LIN {X 0,Y 425.746,Z 248.042,A -85,B 0,C 180,E1 19809.734,E2 19809.734} C_VEL
LIN {X 0,Y 425.285,Z 246.258,A -85,B 0,C 180,E1 19809.199,E2 19809.199} C_VEL
LIN {X 0,Y 425.24,Z 246.07,A -85,B 0,C 180,E1 19805.532,E2 19805.532} C_VEL
LIN {X 0,Y 425.24,Z 246.073,A -85,B 0,C 180,E1 19801.616,E2 19801.616} C_VEL
LIN {X 0,Y 425.257,Z 246.076,A -85,B 0,C 180,E1 19797.978,E2 19797.978} C_VEL
LIN {X 0,Y 425.284,Z 246.063,A -85,B 0,C 180,E1 19794.197,E2 19794.197} C_VEL
LIN {X 0,Y 425.27,Z 246.064,A -85,B 0,C 180,E1 19790.527,E2 19790.527} C_VEL
LIN {X 0,Y 425.247,Z 246.076,A -85,B 0,C 180,E1 19786.749,E2 19786.749} C_VEL
LIN {X 0,Y 425.238,Z 246.075,A -85,B 0,C 180,E1 19783.048,E2 19783.048} C_VEL
LIN {X 0,Y 425.242,Z 246.067,A -85,B 0,C 180,E1 19779.204,E2 19779.204} C_VEL
LIN {X 0,Y 425.274,Z 246.074,A -85,B 0,C 180,E1 19775.556,E2 19775.556} C_VEL
LIN {X 0,Y 425.312,Z 246.344,A -85,B 0,C 180,E1 19773.47,E2 19773.47} C_VEL
LIN {X 0,Y 426.471,Z 249.444,A -85,B 0,C 180,E1 19772.644,E2 19772.644} C_VEL
LIN {X 0,Y 428.836,Z 251.992,A -85,B 0,C 180,E1 19771.751,E2 19771.751} C_VEL
LIN {X 0,Y 430.464,Z 255.45,A -85,B 0,C 180,E1 19770.958,E2 19770.958} C_VEL
LIN {X 0,Y 432.236,Z 257.496,A -85,B 0,C 180,E1 19770.328,E2 19770.328} C_VEL
LIN {X 0,Y 434.45,Z 261.508,A -85,B 0,C 180,E1 19769.428,E2 19769.428} C_VEL
LIN {X 0,Y 435.82,Z 263.65,A -85,B 0,C 180,E1 19768.922,E2 19768.922} C_VEL
LIN {X 0,Y 439.262,Z 269.551,A -85,B 0,C 180,E1 19767.662,E2 19767.662} C_VEL
LIN {X 0,Y 443.697,Z 276.942,A -85,B 0,C 180,E1 19766.178,E2 19766.178} C_VEL
LIN {X 0,Y 451.348,Z 291.113,A -85,B 0,C 180,E1 19763.738,E2 19763.738} C_VEL
LIN {X 0,Y 458.605,Z 305.629,A -85,B 0,C 180,E1 19761.584,E2 19761.584} C_VEL
LIN {X 0,Y 462.483,Z 314.322,A -85,B 0,C 180,E1 19760.454,E2 19760.454} C_VEL
LIN {X 0,Y 461.558,Z 326.532,A -85,B 0,C 180,E1 19759.768,E2 19759.768} C_VEL
LIN {X 0,Y 463.161,Z 344.572,A -85,B 0,C 180,E1 19759.232,E2 19759.232} C_VEL
LIN {X 0,Y 458.976,Z 547.408,A -85,B 0,C 180,E1 19755.792,E2 19755.792} C_VEL
LIN {X 0,Y 456.721,Z 660.808,A -85,B 0,C 180,E1 19753.907,E2 19753.907} C_VEL
LIN {X 0,Y 455.349,Z 683.856,A -85,B 0,C 180,E1 19753.332,E2 19753.332} C_VEL
LIN {X 0,Y 453.601,Z 706.683,A -85,B 0,C 180,E1 19752.542,E2 19752.542} C_VEL
LIN {X 0,Y 451.584,Z 727.107,A -85,B 0,C 180,E1 19751.621,E2 19751.621} C_VEL
LIN {X 0,Y 449.041,Z 749.414,A -85,B 0,C 180,E1 19750.385,E2 19750.385} C_VEL
LIN {X 0,Y 446.38,Z 769.931,A -85,B 0,C 180,E1 19749.005,E2 19749.005} C_VEL
LIN {X 0,Y 443.463,Z 790.74,A -85,B 0,C 180,E1 19747.335,E2 19747.335} C_VEL
LIN {X 0,Y 440.606,Z 810.204,A -85,B 0,C 180,E1 19745.514,E2 19745.514} C_VEL
LIN {X 0,Y 437.767,Z 828.343,A -85,B 0,C 180,E1 19743.523,E2 19743.523} C_VEL
LIN {X 0,Y 434.981,Z 846.538,A -85,B 0,C 180,E1 19741.23,E2 19741.23} C_VEL
LIN {X 0,Y 432.58,Z 862.117,A -85,B 0,C 180,E1 19738.96,E2 19738.96} C_VEL
LIN {X 0,Y 430.192,Z 878.511,A -85,B 0,C 180,E1 19736.204,E2 19736.204} C_VEL
LIN {X 0,Y 428.326,Z 892.284,A -85,B 0,C 180,E1 19733.525,E2 19733.525} C_VEL
LIN {X 0,Y 426.985,Z 902.738,A -85,B 0,C 180,E1 19731.136,E2 19731.136} C_VEL
LIN {X 0,Y 425.868,Z 911.603,A -85,B 0,C 180,E1 19728.619,E2 19728.619} C_VEL
LIN {X 0,Y 424.933,Z 920.642,A -85,B 0,C 180,E1 19725.558,E2 19725.558} C_VEL
LIN {X 0,Y 424.39,Z 927.376,A -85,B 0,C 180,E1 19722.74,E2 19722.74} C_VEL
LIN {X 0,Y 424.071,Z 933.431,A -85,B 0,C 180,E1 19719.498,E2 19719.498} C_VEL
LIN {X 0,Y 423.954,Z 937.12,A -85,B 0,C 180,E1 19716.771,E2 19716.771} C_VEL
LIN {X 0,Y 423.912,Z 939.849,A -85,B 0,C 180,E1 19713.65,E2 19713.65} C_VEL
LIN {X 0,Y 423.907,Z 940.849,A -85,B 0,C 180,E1 19710.945,E2 19710.945} C_VEL
LIN {X 0,Y 423.904,Z 940.658,A -85,B 0,C 180,E1 19707.971,E2 19707.971} C_VEL
LIN {X 0,Y 423.915,Z 938.839,A -85,B 0,C 180,E1 19704.992,E2 19704.992} C_VEL
LIN {X 0,Y 423.995,Z 935.76,A -85,B 0,C 180,E1 19702.07,E2 19702.07} C_VEL
LIN {X 0,Y 424.171,Z 931.079,A -85,B 0,C 180,E1 19699.129,E2 19699.129} C_VEL
LIN {X 0,Y 424.564,Z 925.131,A -85,B 0,C 180,E1 19696.239,E2 19696.239} C_VEL
LIN {X 0,Y 425.27,Z 917.14,A -85,B 0,C 180,E1 19693.189,E2 19693.189} C_VEL
LIN {X 0,Y 426.336,Z 907.927,A -85,B 0,C 180,E1 19690.261,E2 19690.261} C_VEL
LIN {X 0,Y 427.504,Z 898.642,A -85,B 0,C 180,E1 19687.879,E2 19687.879} C_VEL
LIN {X 0,Y 429.068,Z 886.781,A -85,B 0,C 180,E1 19685.343,E2 19685.343} C_VEL
LIN {X 0,Y 431.155,Z 872.227,A -85,B 0,C 180,E1 19682.646,E2 19682.646} C_VEL
LIN {X 0,Y 433.418,Z 857.45,A -85,B 0,C 180,E1 19680.264,E2 19680.264} C_VEL
LIN {X 0,Y 436.1,Z 840.26,A -85,B 0,C 180,E1 19677.864,E2 19677.864} C_VEL
LIN {X 0,Y 438.989,Z 822.381,A -85,B 0,C 180,E1 19675.686,E2 19675.686} C_VEL
LIN {X 0,Y 441.898,Z 803.51,A -85,B 0,C 180,E1 19673.722,E2 19673.722} C_VEL
LIN {X 0,Y 445.127,Z 782.292,A -85,B 0,C 180,E1 19671.83,E2 19671.83} C_VEL
LIN {X 0,Y 447.859,Z 763.075,A -85,B 0,C 180,E1 19670.374,E2 19670.374} C_VEL
LIN {X 0,Y 450.56,Z 741.751,A -85,B 0,C 180,E1 19669.022,E2 19669.022} C_VEL
LIN {X 0,Y 453.012,Z 720.323,A -85,B 0,C 180,E1 19667.9,E2 19667.9} C_VEL
LIN {X 0,Y 455.105,Z 697.951,A -85,B 0,C 180,E1 19666.986,E2 19666.986} C_VEL
LIN {X 0,Y 456.847,Z 674.867,A -85,B 0,C 180,E1 19666.269,E2 19666.269} C_VEL
LIN {X 0,Y 457.896,Z 652.808,A -85,B 0,C 180,E1 19665.792,E2 19665.792} C_VEL
LIN {X 0,Y 462.545,Z 443.623,A -85,B 0,C 180,E1 19662.239,E2 19662.239} C_VEL
LIN {X 0,Y 464.828,Z 341.981,A -85,B 0,C 180,E1 19660.452,E2 19660.452} C_VEL
LIN {X 0,Y 462.948,Z 321.847,A -85,B 0,C 180,E1 19659.812,E2 19659.812} C_VEL
LIN {X 0,Y 463.439,Z 314.532,A -85,B 0,C 180,E1 19659.368,E2 19659.368} C_VEL
LIN {X 0,Y 453.908,Z 296.131,A -85,B 0,C 180,E1 19656.81,E2 19656.81} C_VEL
LIN {X 0,Y 445.163,Z 280.178,A -85,B 0,C 180,E1 19654.316,E2 19654.316} C_VEL
LIN {X 0,Y 436.766,Z 265.785,A -85,B 0,C 180,E1 19651.771,E2 19651.771} C_VEL
LIN {X 0,Y 433.659,Z 260.741,A -85,B 0,C 180,E1 19650.787,E2 19650.787} C_VEL
LIN {X 0,Y 431.047,Z 256.218,A -85,B 0,C 180,E1 19649.915,E2 19649.915} C_VEL
LIN {X 0,Y 428.776,Z 252.669,A -85,B 0,C 180,E1 19649.168,E2 19649.168} C_VEL
LIN {X 0,Y 428.12,Z 251.254,A -85,B 0,C 180,E1 19648.911,E2 19648.911} C_VEL
LIN {X 0,Y 425.814,Z 248.061,A -85,B 0,C 180,E1 19648.163,E2 19648.163} C_VEL
LIN {X 0,Y 425.317,Z 246.402,A -85,B 0,C 180,E1 19647.817,E2 19647.817} C_VEL
LIN {X 0,Y 425.298,Z 246.06,A -85,B 0,C 180,E1 19646.531,E2 19646.531} C_VEL
LIN {X 0,Y 425.27,Z 246.06,A -85,B 0,C 180,E1 19642.826,E2 19642.826} C_VEL
LIN {X 0,Y 425.263,Z 246.059,A -85,B 0,C 180,E1 19639.06,E2 19639.06} C_VEL
LIN {X 0,Y 425.268,Z 246.059,A -85,B 0,C 180,E1 19635.268,E2 19635.268} C_VEL
LIN {X 0,Y 425.288,Z 246.064,A -85,B 0,C 180,E1 19631.528,E2 19631.528} C_VEL
LIN {X 0,Y 425.312,Z 246.067,A -85,B 0,C 180,E1 19627.701,E2 19627.701} C_VEL
LIN {X 0,Y 425.316,Z 246.067,A -85,B 0,C 180,E1 19623.91,E2 19623.91} C_VEL
LIN {X 0,Y 425.314,Z 246.052,A -85,B 0,C 180,E1 19620,E2 19620} C_VEL
LIN {X 0,Y 425.292,Z 246.048,A -85,B 0,C 180,E1 19616.226,E2 19616.226} C_VEL
LIN {X 0,Y 425.286,Z 246.06,A -85,B 0,C 180,E1 19612.435,E2 19612.435} C_VEL
LIN {X 0,Y 425.291,Z 246.07,A -85,B 0,C 180,E1 19608.611,E2 19608.611} C_VEL
LIN {X 0,Y 425.298,Z 246.059,A -85,B 0,C 180,E1 19604.734,E2 19604.734} C_VEL
LIN {X 0,Y 425.312,Z 246.042,A -85,B 0,C 180,E1 19600.921,E2 19600.921} C_VEL
LIN {X 0,Y 425.322,Z 246.059,A -85,B 0,C 180,E1 19597.031,E2 19597.031} C_VEL
LIN {X 0,Y 425.319,Z 246.07,A -85,B 0,C 180,E1 19593.17,E2 19593.17} C_VEL
LIN {X 0,Y 425.32,Z 246.05,A -85,B 0,C 180,E1 19589.328,E2 19589.328} C_VEL
LIN {X 0,Y 425.312,Z 246.047,A -85,B 0,C 180,E1 19585.49,E2 19585.49} C_VEL
LIN {X 0,Y 425.309,Z 246.056,A -85,B 0,C 180,E1 19581.638,E2 19581.638} C_VEL
LIN {X 0,Y 425.309,Z 246.071,A -85,B 0,C 180,E1 19577.752,E2 19577.752} C_VEL
LIN {X 0,Y 425.313,Z 246.067,A -85,B 0,C 180,E1 19573.91,E2 19573.91} C_VEL
LIN {X 0,Y 425.319,Z 246.06,A -85,B 0,C 180,E1 19570.102,E2 19570.102} C_VEL
LIN {X 0,Y 425.309,Z 246.057,A -85,B 0,C 180,E1 19566.26,E2 19566.26} C_VEL
LIN {X 0,Y 425.303,Z 246.058,A -85,B 0,C 180,E1 19562.414,E2 19562.414} C_VEL
LIN {X 0,Y 425.303,Z 246.064,A -85,B 0,C 180,E1 19558.506,E2 19558.506} C_VEL
LIN {X 0,Y 425.333,Z 246.177,A -85,B 0,C 180,E1 19555.332,E2 19555.332} C_VEL
LIN {X 0,Y 425.718,Z 247.757,A -85,B 0,C 180,E1 19554.966,E2 19554.966} C_VEL
LIN {X 0,Y 427.723,Z 250.874,A -85,B 0,C 180,E1 19554.264,E2 19554.264} C_VEL
LIN {X 0,Y 430.512,Z 255.747,A -85,B 0,C 180,E1 19553.256,E2 19553.256} C_VEL
LIN {X 0,Y 438.381,Z 270.408,A -85,B 0,C 180,E1 19550.488,E2 19550.488} C_VEL
LIN {X 0,Y 446.356,Z 286.148,A -85,B 0,C 180,E1 19547.824,E2 19547.824} C_VEL
LIN {X 0,Y 454.871,Z 304.797,A -85,B 0,C 180,E1 19545.034,E2 19545.034} C_VEL
LIN {X 0,Y 455.747,Z 306.894,A -85,B 0,C 180,E1 19544.745,E2 19544.745} C_VEL
LIN {X 0,Y 450.346,Z 360.908,A -85,B 0,C 180,E1 19540.814,E2 19540.814} C_VEL
LIN {X 0,Y 448.535,Z 380.257,A -85,B 0,C 180,E1 19539.42,E2 19539.42} C_VEL
LIN {X 0,Y 447.096,Z 387.162,A -85,B 0,C 180,E1 19539.008,E2 19539.008} C_VEL
LIN {X 0,Y 442.737,Z 400.415,A -85,B 0,C 180,E1 19538.506,E2 19538.506} C_VEL
LIN {X 0,Y 441.127,Z 408.875,A -85,B 0,C 180,E1 19538.25,E2 19538.25} C_VEL
LIN {X 0,Y 441.203,Z 413.135,A -85,B 0,C 180,E1 19538.111,E2 19538.111} C_VEL
LIN {X 0,Y 444.354,Z 443.954,A -85,B 0,C 180,E1 19537.096,E2 19537.096} C_VEL
LIN {X 0,Y 438.364,Z 627.681,A -85,B 0,C 180,E1 19533.716,E2 19533.716} C_VEL
LIN {X 0,Y 437.228,Z 648.183,A -85,B 0,C 180,E1 19533.157,E2 19533.157} C_VEL
LIN {X 0,Y 435.704,Z 667.803,A -85,B 0,C 180,E1 19532.369,E2 19532.369} C_VEL
LIN {X 0,Y 433.951,Z 686.035,A -85,B 0,C 180,E1 19531.388,E2 19531.388} C_VEL
LIN {X 0,Y 431.933,Z 703.655,A -85,B 0,C 180,E1 19530.185,E2 19530.185} C_VEL
LIN {X 0,Y 429.819,Z 720.048,A -85,B 0,C 180,E1 19528.802,E2 19528.802} C_VEL
LIN {X 0,Y 427.62,Z 735.774,A -85,B 0,C 180,E1 19527.187,E2 19527.187} C_VEL
LIN {X 0,Y 425.516,Z 750.047,A -85,B 0,C 180,E1 19525.419,E2 19525.419} C_VEL
LIN {X 0,Y 423.41,Z 763.852,A -85,B 0,C 180,E1 19523.357,E2 19523.357} C_VEL
LIN {X 0,Y 421.564,Z 776.1,A -85,B 0,C 180,E1 19521.133,E2 19521.133} C_VEL
LIN {X 0,Y 420.097,Z 786.256,A -85,B 0,C 180,E1 19518.886,E2 19518.886} C_VEL
LIN {X 0,Y 418.901,Z 795.102,A -85,B 0,C 180,E1 19516.474,E2 19516.474} C_VEL
LIN {X 0,Y 418.026,Z 802.528,A -85,B 0,C 180,E1 19513.893,E2 19513.893} C_VEL
LIN {X 0,Y 417.451,Z 808.152,A -85,B 0,C 180,E1 19511.281,E2 19511.281} C_VEL
LIN {X 0,Y 417.118,Z 812.066,A -85,B 0,C 180,E1 19508.634,E2 19508.634} C_VEL
LIN {X 0,Y 416.979,Z 814.309,A -85,B 0,C 180,E1 19505.945,E2 19505.945} C_VEL
LIN {X 0,Y 416.98,Z 814.86,A -85,B 0,C 180,E1 19503.207,E2 19503.207} C_VEL
LIN {X 0,Y 417.097,Z 813.743,A -85,B 0,C 180,E1 19500.568,E2 19500.568} C_VEL
LIN {X 0,Y 417.382,Z 810.908,A -85,B 0,C 180,E1 19497.874,E2 19497.874} C_VEL
LIN {X 0,Y 417.896,Z 806.506,A -85,B 0,C 180,E1 19495.291,E2 19495.291} C_VEL
LIN {X 0,Y 418.699,Z 800.222,A -85,B 0,C 180,E1 19492.661,E2 19492.661} C_VEL
LIN {X 0,Y 419.829,Z 792.38,A -85,B 0,C 180,E1 19490.162,E2 19490.162} C_VEL
LIN {X 0,Y 421.33,Z 782.898,A -85,B 0,C 180,E1 19487.765,E2 19487.765} C_VEL
LIN {X 0,Y 423.183,Z 771.548,A -85,B 0,C 180,E1 19485.437,E2 19485.437} C_VEL
LIN {X 0,Y 425.264,Z 759.169,A -85,B 0,C 180,E1 19483.355,E2 19483.355} C_VEL
LIN {X 0,Y 427.517,Z 745.456,A -85,B 0,C 180,E1 19481.441,E2 19481.441} C_VEL
LIN {X 0,Y 429.933,Z 730.11,A -85,B 0,C 180,E1 19479.669,E2 19479.669} C_VEL
LIN {X 0,Y 432.297,Z 713.987,A -85,B 0,C 180,E1 19478.136,E2 19478.136} C_VEL
LIN {X 0,Y 434.583,Z 696.897,A -85,B 0,C 180,E1 19476.811,E2 19476.811} C_VEL
LIN {X 0,Y 436.755,Z 678.012,A -85,B 0,C 180,E1 19475.643,E2 19475.643} C_VEL
LIN {X 0,Y 438.614,Z 658.486,A -85,B 0,C 180,E1 19474.721,E2 19474.721} C_VEL
LIN {X 0,Y 440.085,Z 638.517,A -85,B 0,C 180,E1 19474.044,E2 19474.044} C_VEL
LIN {X 0,Y 441.319,Z 612.376,A -85,B 0,C 180,E1 19473.474,E2 19473.474} C_VEL
LIN {X 0,Y 447.993,Z 443.231,A -85,B 0,C 180,E1 19470.231,E2 19470.231} C_VEL
LIN {X 0,Y 443.246,Z 397.447,A -85,B 0,C 180,E1 19468.528,E2 19468.528} C_VEL
LIN {X 0,Y 449.564,Z 341.197,A -85,B 0,C 180,E1 19464.365,E2 19464.365} C_VEL
LIN {X 0,Y 452.772,Z 314.572,A -85,B 0,C 180,E1 19462.357,E2 19462.357} C_VEL
LIN {X 0,Y 445.764,Z 299.009,A -85,B 0,C 180,E1 19459.797,E2 19459.797} C_VEL
LIN {X 0,Y 439.03,Z 285.264,A -85,B 0,C 180,E1 19457.221,E2 19457.221} C_VEL
LIN {X 0,Y 433.996,Z 275.992,A -85,B 0,C 180,E1 19455.226,E2 19455.226} C_VEL
LIN {X 0,Y 429.591,Z 267.882,A -85,B 0,C 180,E1 19453.321,E2 19453.321} C_VEL
LIN {X 0,Y 427.293,Z 263.861,A -85,B 0,C 180,E1 19452.294,E2 19452.294} C_VEL
LIN {X 0,Y 424.471,Z 259.342,A -85,B 0,C 180,E1 19450.999,E2 19450.999} C_VEL
LIN {X 0,Y 423.749,Z 257.833,A -85,B 0,C 180,E1 19450.605,E2 19450.605} C_VEL
LIN {X 0,Y 421.453,Z 254.749,A -85,B 0,C 180,E1 19449.559,E2 19449.559} C_VEL
LIN {X 0,Y 420.354,Z 252.378,A -85,B 0,C 180,E1 19448.894,E2 19448.894} C_VEL
LIN {X 0,Y 417.951,Z 249.368,A -85,B 0,C 180,E1 19447.698,E2 19447.698} C_VEL
LIN {X 0,Y 417.359,Z 247.266,A -85,B 0,C 180,E1 19447.017,E2 19447.017} C_VEL
LIN {X 0,Y 417.304,Z 247.062,A -85,B 0,C 180,E1 19443.296,E2 19443.296} C_VEL
LIN {X 0,Y 417.299,Z 247.055,A -85,B 0,C 180,E1 19439.588,E2 19439.588} C_VEL
LIN {X 0,Y 417.317,Z 247.06,A -85,B 0,C 180,E1 19435.878,E2 19435.878} C_VEL
LIN {X 0,Y 417.351,Z 247.061,A -85,B 0,C 180,E1 19432.151,E2 19432.151} C_VEL
LIN {X 0,Y 417.344,Z 247.051,A -85,B 0,C 180,E1 19428.25,E2 19428.25} C_VEL
LIN {X 0,Y 417.313,Z 247.055,A -85,B 0,C 180,E1 19424.576,E2 19424.576} C_VEL
LIN {X 0,Y 417.302,Z 247.068,A -85,B 0,C 180,E1 19420.837,E2 19420.837} C_VEL
LIN {X 0,Y 417.299,Z 247.057,A -85,B 0,C 180,E1 19416.931,E2 19416.931} C_VEL
LIN {X 0,Y 417.389,Z 247.388,A -85,B 0,C 180,E1 19415.626,E2 19415.626} C_VEL
LIN {X 0,Y 418.847,Z 250.873,A -85,B 0,C 180,E1 19414.552,E2 19414.552} C_VEL
LIN {X 0,Y 421.017,Z 253.041,A -85,B 0,C 180,E1 19413.634,E2 19413.634} C_VEL
LIN {X 0,Y 422.761,Z 256.674,A -85,B 0,C 180,E1 19412.689,E2 19412.689} C_VEL
LIN {X 0,Y 424.463,Z 258.414,A -85,B 0,C 180,E1 19412.044,E2 19412.044} C_VEL
LIN {X 0,Y 426.407,Z 262.256,A -85,B 0,C 180,E1 19411.116,E2 19411.116} C_VEL
LIN {X 0,Y 428.077,Z 264.553,A -85,B 0,C 180,E1 19410.473,E2 19410.473} C_VEL
LIN {X 0,Y 431.649,Z 270.612,A -85,B 0,C 180,E1 19409.054,E2 19409.054} C_VEL
LIN {X 0,Y 434.736,Z 275.889,A -85,B 0,C 180,E1 19407.908,E2 19407.908} C_VEL
LIN {X 0,Y 439.42,Z 284.026,A -85,B 0,C 180,E1 19406.275,E2 19406.275} C_VEL
LIN {X 0,Y 446.627,Z 297.494,A -85,B 0,C 180,E1 19403.93,E2 19403.93} C_VEL
LIN {X 0,Y 454.625,Z 313.832,A -85,B 0,C 180,E1 19401.508,E2 19401.508} C_VEL
LIN {X 0,Y 456.377,Z 317.895,A -85,B 0,C 180,E1 19400.979,E2 19400.979} C_VEL
LIN {X 0,Y 455.6,Z 327.719,A -85,B 0,C 180,E1 19400.423,E2 19400.423} C_VEL
LIN {X 0,Y 457.148,Z 345.946,A -85,B 0,C 180,E1 19399.874,E2 19399.874} C_VEL
LIN {X 0,Y 452.657,Z 548.561,A -85,B 0,C 180,E1 19396.397,E2 19396.397} C_VEL
LIN {X 0,Y 450.302,Z 660.702,A -85,B 0,C 180,E1 19394.514,E2 19394.514} C_VEL
LIN {X 0,Y 448.874,Z 683.498,A -85,B 0,C 180,E1 19393.94,E2 19393.94} C_VEL
LIN {X 0,Y 447.112,Z 705.489,A -85,B 0,C 180,E1 19393.178,E2 19393.178} C_VEL
LIN {X 0,Y 444.92,Z 726.669,A -85,B 0,C 180,E1 19392.214,E2 19392.214} C_VEL
LIN {X 0,Y 442.26,Z 748.917,A -85,B 0,C 180,E1 19390.965,E2 19390.965} C_VEL
LIN {X 0,Y 439.616,Z 768.347,A -85,B 0,C 180,E1 19389.646,E2 19389.646} C_VEL
LIN {X 0,Y 436.514,Z 789.369,A -85,B 0,C 180,E1 19387.951,E2 19387.951} C_VEL
LIN {X 0,Y 433.506,Z 808.88,A -85,B 0,C 180,E1 19386.105,E2 19386.105} C_VEL
LIN {X 0,Y 430.444,Z 827.459,A -85,B 0,C 180,E1 19384.04,E2 19384.04} C_VEL
LIN {X 0,Y 427.554,Z 845.389,A -85,B 0,C 180,E1 19381.745,E2 19381.745} C_VEL
LIN {X 0,Y 424.982,Z 861.229,A -85,B 0,C 180,E1 19379.398,E2 19379.398} C_VEL
LIN {X 0,Y 422.575,Z 876.944,A -85,B 0,C 180,E1 19376.714,E2 19376.714} C_VEL
LIN {X 0,Y 420.67,Z 890.112,A -85,B 0,C 180,E1 19374.119,E2 19374.119} C_VEL
LIN {X 0,Y 419.03,Z 902.525,A -85,B 0,C 180,E1 19371.264,E2 19371.264} C_VEL
LIN {X 0,Y 417.811,Z 913.155,A -85,B 0,C 180,E1 19368.413,E2 19368.413} C_VEL
LIN {X 0,Y 416.993,Z 920.994,A -85,B 0,C 180,E1 19365.719,E2 19365.719} C_VEL
LIN {X 0,Y 416.424,Z 927.604,A -85,B 0,C 180,E1 19362.882,E2 19362.882} C_VEL
LIN {X 0,Y 416.085,Z 933.432,A -85,B 0,C 180,E1 19359.682,E2 19359.682} C_VEL
LIN {X 0,Y 415.958,Z 937.12,A -85,B 0,C 180,E1 19356.901,E2 19356.901} C_VEL
LIN {X 0,Y 415.913,Z 939.848,A -85,B 0,C 180,E1 19353.72,E2 19353.72} C_VEL
LIN {X 0,Y 415.908,Z 940.848,A -85,B 0,C 180,E1 19350.963,E2 19350.963} C_VEL
LIN {X 0,Y 415.905,Z 940.658,A -85,B 0,C 180,E1 19347.932,E2 19347.932} C_VEL
LIN {X 0,Y 415.918,Z 938.839,A -85,B 0,C 180,E1 19344.896,E2 19344.896} C_VEL
LIN {X 0,Y 415.997,Z 935.839,A -85,B 0,C 180,E1 19341.985,E2 19341.985} C_VEL
LIN {X 0,Y 416.195,Z 931.079,A -85,B 0,C 180,E1 19338.918,E2 19338.918} C_VEL
LIN {X 0,Y 416.63,Z 925.131,A -85,B 0,C 180,E1 19335.971,E2 19335.971} C_VEL
LIN {X 0,Y 417.381,Z 917.24,A -85,B 0,C 180,E1 19332.906,E2 19332.906} C_VEL
LIN {X 0,Y 418.133,Z 910.125,A -85,B 0,C 180,E1 19330.73,E2 19330.73} C_VEL
LIN {X 0,Y 419.563,Z 898.531,A -85,B 0,C 180,E1 19327.732,E2 19327.732} C_VEL
LIN {X 0,Y 421.251,Z 886.306,A -85,B 0,C 180,E1 19325.052,E2 19325.052} C_VEL
LIN {X 0,Y 423.579,Z 870.879,A -85,B 0,C 180,E1 19322.134,E2 19322.134} C_VEL
LIN {X 0,Y 426.154,Z 855.056,A -85,B 0,C 180,E1 19319.549,E2 19319.549} C_VEL
LIN {X 0,Y 428.952,Z 838.143,A -85,B 0,C 180,E1 19317.183,E2 19317.183} C_VEL
LIN {X 0,Y 432.022,Z 820.024,A -85,B 0,C 180,E1 19314.972,E2 19314.972} C_VEL
LIN {X 0,Y 435.01,Z 801.745,A -85,B 0,C 180,E1 19313.054,E2 19313.054} C_VEL
LIN {X 0,Y 438.266,Z 781.378,A -85,B 0,C 180,E1 19311.225,E2 19311.225} C_VEL
LIN {X 0,Y 441.2,Z 761.669,A -85,B 0,C 180,E1 19309.721,E2 19309.721} C_VEL
LIN {X 0,Y 444.003,Z 740.398,A -85,B 0,C 180,E1 19308.369,E2 19308.369} C_VEL
LIN {X 0,Y 446.561,Z 719.196,A -85,B 0,C 180,E1 19307.257,E2 19307.257} C_VEL
LIN {X 0,Y 448.7,Z 697.195,A -85,B 0,C 180,E1 19306.355,E2 19306.355} C_VEL
LIN {X 0,Y 450.523,Z 673.886,A -85,B 0,C 180,E1 19305.632,E2 19305.632} C_VEL
LIN {X 0,Y 451.59,Z 651.951,A -85,B 0,C 180,E1 19305.157,E2 19305.157} C_VEL
LIN {X 0,Y 456.42,Z 445.423,A -85,B 0,C 180,E1 19301.618,E2 19301.618} C_VEL
LIN {X 0,Y 458.869,Z 343.258,A -85,B 0,C 180,E1 19299.802,E2 19299.802} C_VEL
LIN {X 0,Y 457.028,Z 322.48,A -85,B 0,C 180,E1 19299.128,E2 19299.128} C_VEL
LIN {X 0,Y 457.276,Z 318.362,A -85,B 0,C 180,E1 19298.869,E2 19298.869} C_VEL
LIN {X 0,Y 447.037,Z 298.453,A -85,B 0,C 180,E1 19296.032,E2 19296.032} C_VEL
LIN {X 0,Y 437.188,Z 280.817,A -85,B 0,C 180,E1 19293.134,E2 19293.134} C_VEL
LIN {X 0,Y 429.413,Z 267.492,A -85,B 0,C 180,E1 19290.659,E2 19290.659} C_VEL
LIN {X 0,Y 425.973,Z 261.973,A -85,B 0,C 180,E1 19289.533,E2 19289.533} C_VEL
LIN {X 0,Y 423.066,Z 257.122,A -85,B 0,C 180,E1 19288.516,E2 19288.516} C_VEL
LIN {X 0,Y 420.906,Z 253.592,A -85,B 0,C 180,E1 19287.749,E2 19287.749} C_VEL
LIN {X 0,Y 420.239,Z 252.312,A -85,B 0,C 180,E1 19287.489,E2 19287.489} C_VEL
LIN {X 0,Y 417.966,Z 249.302,A -85,B 0,C 180,E1 19286.727,E2 19286.727} C_VEL
LIN {X 0,Y 417.405,Z 247.325,A -85,B 0,C 180,E1 19286.305,E2 19286.305} C_VEL
LIN {X 0,Y 417.352,Z 247.043,A -85,B 0,C 180,E1 19282.54,E2 19282.54} C_VEL
LIN {X 0,Y 417.331,Z 247.045,A -85,B 0,C 180,E1 19278.849,E2 19278.849} C_VEL
LIN {X 0,Y 417.326,Z 247.046,A -85,B 0,C 180,E1 19275.084,E2 19275.084} C_VEL
LIN {X 0,Y 417.333,Z 247.048,A -85,B 0,C 180,E1 19271.19,E2 19271.19} C_VEL
LIN {X 0,Y 417.35,Z 247.057,A -85,B 0,C 180,E1 19267.434,E2 19267.434} C_VEL
LIN {X 0,Y 417.377,Z 247.06,A -85,B 0,C 180,E1 19263.709,E2 19263.709} C_VEL
LIN {X 0,Y 417.386,Z 247.043,A -85,B 0,C 180,E1 19259.726,E2 19259.726} C_VEL
LIN {X 0,Y 417.371,Z 247.034,A -85,B 0,C 180,E1 19255.879,E2 19255.879} C_VEL
LIN {X 0,Y 417.357,Z 247.041,A -85,B 0,C 180,E1 19252.152,E2 19252.152} C_VEL
LIN {X 0,Y 417.354,Z 247.061,A -85,B 0,C 180,E1 19248.251,E2 19248.251} C_VEL
LIN {X 0,Y 417.354,Z 247.053,A -85,B 0,C 180,E1 19244.384,E2 19244.384} C_VEL
LIN {X 0,Y 417.358,Z 247.032,A -85,B 0,C 180,E1 19240.55,E2 19240.55} C_VEL
LIN {X 0,Y 417.374,Z 247.044,A -85,B 0,C 180,E1 19236.718,E2 19236.718} C_VEL
LIN {X 0,Y 417.38,Z 247.056,A -85,B 0,C 180,E1 19232.772,E2 19232.772} C_VEL
LIN {X 0,Y 417.38,Z 247.048,A -85,B 0,C 180,E1 19228.84,E2 19228.84} C_VEL
LIN {X 0,Y 417.373,Z 247.036,A -85,B 0,C 180,E1 19224.905,E2 19224.905} C_VEL
LIN {X 0,Y 417.377,Z 247.035,A -85,B 0,C 180,E1 19221.125,E2 19221.125} C_VEL
LIN {X 0,Y 417.375,Z 247.05,A -85,B 0,C 180,E1 19217.317,E2 19217.317} C_VEL
LIN {X 0,Y 417.376,Z 247.06,A -85,B 0,C 180,E1 19213.436,E2 19213.436} C_VEL
LIN {X 0,Y 417.375,Z 247.056,A -85,B 0,C 180,E1 19209.524,E2 19209.524} C_VEL
LIN {X 0,Y 417.377,Z 247.056,A -85,B 0,C 180,E1 19205.601,E2 19205.601} C_VEL
LIN {X 0,Y 417.379,Z 247.058,A -85,B 0,C 180,E1 19201.644,E2 19201.644} C_VEL
LIN {X 0,Y 417.379,Z 247.058,A -85,B 0,C 180,E1 19197.85,E2 19197.85} C_VEL
LIN {X 0,Y 417.414,Z 247.375,A -85,B 0,C 180,E1 19196.655,E2 19196.655} C_VEL
LIN {X 0,Y 418.952,Z 250.911,A -85,B 0,C 180,E1 19195.879,E2 19195.879} C_VEL
LIN {X 0,Y 420.313,Z 252.613,A -85,B 0,C 180,E1 19195.429,E2 19195.429} C_VEL
LIN {X 0,Y 422.341,Z 256.501,A -85,B 0,C 180,E1 19194.623,E2 19194.623} C_VEL
LIN {X 0,Y 426.288,Z 263.546,A -85,B 0,C 180,E1 19193.159,E2 19193.159} C_VEL
LIN {X 0,Y 430.93,Z 272.023,A -85,B 0,C 180,E1 19191.503,E2 19191.503} C_VEL
LIN {X 0,Y 439.077,Z 287.979,A -85,B 0,C 180,E1 19188.685,E2 19188.685} C_VEL
LIN {X 0,Y 447.369,Z 305.864,A -85,B 0,C 180,E1 19185.897,E2 19185.897} C_VEL
LIN {X 0,Y 449.37,Z 310.917,A -85,B 0,C 180,E1 19185.19,E2 19185.19} C_VEL
LIN {X 0,Y 443.738,Z 364.65,A -85,B 0,C 180,E1 19181.241,E2 19181.241} C_VEL
LIN {X 0,Y 440.135,Z 403.413,A -85,B 0,C 180,E1 19178.447,E2 19178.447} C_VEL
LIN {X 0,Y 441.203,Z 413.135,A -85,B 0,C 180,E1 19178.111,E2 19178.111} C_VEL
LIN {X 0,Y 441.37,Z 420.755,A -85,B 0,C 180,E1 19177.925,E2 19177.925} C_VEL
LIN {X 0,Y 439.742,Z 434.037,A -85,B 0,C 180,E1 19177.811,E2 19177.811} C_VEL
LIN {X 0,Y 438.085,Z 447.405,A -85,B 0,C 180,E1 19177.698,E2 19177.698} C_VEL
LIN {X 0,Y 438.034,Z 448.519,A -85,B 0,C 180,E1 19177.679,E2 19177.679} C_VEL
LIN {X 0,Y 431.823,Z 628.659,A -85,B 0,C 180,E1 19174.313,E2 19174.313} C_VEL
LIN {X 0,Y 430.63,Z 648.95,A -85,B 0,C 180,E1 19173.746,E2 19173.746} C_VEL
LIN {X 0,Y 429.077,Z 667.933,A -85,B 0,C 180,E1 19172.973,E2 19172.973} C_VEL
LIN {X 0,Y 427.179,Z 686.776,A -85,B 0,C 180,E1 19171.948,E2 19171.948} C_VEL
LIN {X 0,Y 425.079,Z 704.215,A -85,B 0,C 180,E1 19170.743,E2 19170.743} C_VEL
LIN {X 0,Y 422.722,Z 721.541,A -85,B 0,C 180,E1 19169.256,E2 19169.256} C_VEL
LIN {X 0,Y 420.411,Z 737.173,A -85,B 0,C 180,E1 19167.616,E2 19167.616} C_VEL
LIN {X 0,Y 418.093,Z 752.014,A -85,B 0,C 180,E1 19165.732,E2 19165.732} C_VEL
LIN {X 0,Y 415.899,Z 765.561,A -85,B 0,C 180,E1 19163.652,E2 19163.652} C_VEL
LIN {X 0,Y 414.062,Z 777.004,A -85,B 0,C 180,E1 19161.531,E2 19161.531} C_VEL
LIN {X 0,Y 412.398,Z 787.775,A -85,B 0,C 180,E1 19159.101,E2 19159.101} C_VEL
LIN {X 0,Y 411.114,Z 796.661,A -85,B 0,C 180,E1 19156.608,E2 19156.608} C_VEL
LIN {X 0,Y 410.195,Z 803.915,A -85,B 0,C 180,E1 19154.013,E2 19154.013} C_VEL
LIN {X 0,Y 409.58,Z 809.487,A -85,B 0,C 180,E1 19151.351,E2 19151.351} C_VEL
LIN {X 0,Y 409.222,Z 813.358,A -85,B 0,C 180,E1 19148.652,E2 19148.652} C_VEL
LIN {X 0,Y 409.077,Z 815.484,A -85,B 0,C 180,E1 19146.065,E2 19146.065} C_VEL
LIN {X 0,Y 409.075,Z 816.099,A -85,B 0,C 180,E1 19143.275,E2 19143.275} C_VEL
LIN {X 0,Y 409.199,Z 815.053,A -85,B 0,C 180,E1 19140.587,E2 19140.587} C_VEL
LIN {X 0,Y 409.504,Z 812.297,A -85,B 0,C 180,E1 19137.843,E2 19137.843} C_VEL
LIN {X 0,Y 410.098,Z 807.653,A -85,B 0,C 180,E1 19135.046,E2 19135.046} C_VEL
LIN {X 0,Y 410.975,Z 801.346,A -85,B 0,C 180,E1 19132.365,E2 19132.365} C_VEL
LIN {X 0,Y 412.205,Z 793.488,A -85,B 0,C 180,E1 19129.82,E2 19129.82} C_VEL
LIN {X 0,Y 413.853,Z 783.827,A -85,B 0,C 180,E1 19127.34,E2 19127.34} C_VEL
LIN {X 0,Y 415.809,Z 772.654,A -85,B 0,C 180,E1 19125.015,E2 19125.015} C_VEL
LIN {X 0,Y 418.066,Z 760.036,A -85,B 0,C 180,E1 19122.862,E2 19122.862} C_VEL
LIN {X 0,Y 420.515,Z 746.004,A -85,B 0,C 180,E1 19120.881,E2 19120.881} C_VEL
LIN {X 0,Y 423.095,Z 730.551,A -85,B 0,C 180,E1 19119.079,E2 19119.079} C_VEL
LIN {X 0,Y 425.573,Z 714.54,A -85,B 0,C 180,E1 19117.542,E2 19117.542} C_VEL
LIN {X 0,Y 428.076,Z 696.683,A -85,B 0,C 180,E1 19116.15,E2 19116.15} C_VEL
LIN {X 0,Y 430.254,Z 678.643,A -85,B 0,C 180,E1 19115.029,E2 19115.029} C_VEL
LIN {X 0,Y 432.215,Z 659.052,A -85,B 0,C 180,E1 19114.092,E2 19114.092} C_VEL
LIN {X 0,Y 433.772,Z 639.02,A -85,B 0,C 180,E1 19113.403,E2 19113.403} C_VEL
LIN {X 0,Y 435.106,Z 612.36,A -85,B 0,C 180,E1 19112.811,E2 19112.811} C_VEL
LIN {X 0,Y 442.095,Z 444.437,A -85,B 0,C 180,E1 19109.544,E2 19109.544} C_VEL
LIN {X 0,Y 437.284,Z 395.999,A -85,B 0,C 180,E1 19107.692,E2 19107.692} C_VEL
LIN {X 0,Y 443.804,Z 341.368,A -85,B 0,C 180,E1 19103.596,E2 19103.596} C_VEL
LIN {X 0,Y 446.749,Z 318.733,A -85,B 0,C 180,E1 19101.878,E2 19101.878} C_VEL
LIN {X 0,Y 439.83,Z 303.093,A -85,B 0,C 180,E1 19099.245,E2 19099.245} C_VEL
LIN {X 0,Y 432.476,Z 288.05,A -85,B 0,C 180,E1 19096.313,E2 19096.313} C_VEL
LIN {X 0,Y 425.214,Z 274.503,A -85,B 0,C 180,E1 19093.184,E2 19093.184} C_VEL
LIN {X 0,Y 421.759,Z 268.82,A -85,B 0,C 180,E1 19091.625,E2 19091.625} C_VEL
LIN {X 0,Y 419.134,Z 264.174,A -85,B 0,C 180,E1 19090.306,E2 19090.306} C_VEL
LIN {X 0,Y 416.785,Z 260.475,A -85,B 0,C 180,E1 19089.11,E2 19089.11} C_VEL
LIN {X 0,Y 416.143,Z 259.087,A -85,B 0,C 180,E1 19088.706,E2 19088.706} C_VEL
LIN {X 0,Y 413.779,Z 256.056,A -85,B 0,C 180,E1 19087.497,E2 19087.497} C_VEL
LIN {X 0,Y 412.586,Z 253.49,A -85,B 0,C 180,E1 19086.679,E2 19086.679} C_VEL
LIN {X 0,Y 410.195,Z 250.722,A -85,B 0,C 180,E1 19085.314,E2 19085.314} C_VEL
LIN {X 0,Y 409.458,Z 248.402,A -85,B 0,C 180,E1 19084.481,E2 19084.481} C_VEL
LIN {X 0,Y 409.409,Z 248.039,A -85,B 0,C 180,E1 19082.519,E2 19082.519} C_VEL
LIN {X 0,Y 409.407,Z 248.046,A -85,B 0,C 180,E1 19078.6,E2 19078.6} C_VEL
LIN {X 0,Y 409.388,Z 248.046,A -85,B 0,C 180,E1 19074.674,E2 19074.674} C_VEL
LIN {X 0,Y 409.364,Z 248.043,A -85,B 0,C 180,E1 19071.006,E2 19071.006} C_VEL
LIN {X 0,Y 409.36,Z 248.048,A -85,B 0,C 180,E1 19067.157,E2 19067.157} C_VEL
LIN {X 0,Y 409.364,Z 248.054,A -85,B 0,C 180,E1 19063.249,E2 19063.249} C_VEL
LIN {X 0,Y 409.374,Z 248.043,A -85,B 0,C 180,E1 19059.408,E2 19059.408} C_VEL
LIN {X 0,Y 409.435,Z 248.377,A -85,B 0,C 180,E1 19058.261,E2 19058.261} C_VEL
LIN {X 0,Y 410.942,Z 251.914,A -85,B 0,C 180,E1 19056.938,E2 19056.938} C_VEL
LIN {X 0,Y 413.327,Z 254.43,A -85,B 0,C 180,E1 19055.717,E2 19055.717} C_VEL
LIN {X 0,Y 415.17,Z 258.026,A -85,B 0,C 180,E1 19054.616,E2 19054.616} C_VEL
LIN {X 0,Y 416.963,Z 260.022,A -85,B 0,C 180,E1 19053.818,E2 19053.818} C_VEL
LIN {X 0,Y 419.068,Z 263.866,A -85,B 0,C 180,E1 19052.736,E2 19052.736} C_VEL
LIN {X 0,Y 420.345,Z 265.438,A -85,B 0,C 180,E1 19052.211,E2 19052.211} C_VEL
LIN {X 0,Y 422.698,Z 269.485,A -85,B 0,C 180,E1 19051.148,E2 19051.148} C_VEL
LIN {X 0,Y 423.949,Z 271.535,A -85,B 0,C 180,E1 19050.623,E2 19050.623} C_VEL
LIN {X 0,Y 429.224,Z 280.305,A -85,B 0,C 180,E1 19048.547,E2 19048.547} C_VEL
LIN {X 0,Y 436.3,Z 292.991,A -85,B 0,C 180,E1 19046.001,E2 19046.001} C_VEL
LIN {X 0,Y 443.044,Z 306.28,A -85,B 0,C 180,E1 19043.752,E2 19043.752} C_VEL
LIN {X 0,Y 450.299,Z 321.522,A -85,B 0,C 180,E1 19041.515,E2 19041.515} C_VEL
LIN {X 0,Y 449.732,Z 328.711,A -85,B 0,C 180,E1 19041.109,E2 19041.109} C_VEL
LIN {X 0,Y 451.225,Z 347.241,A -85,B 0,C 180,E1 19040.538,E2 19040.538} C_VEL
LIN {X 0,Y 446.465,Z 547.442,A -85,B 0,C 180,E1 19037.061,E2 19037.061} C_VEL
LIN {X 0,Y 443.944,Z 660.313,A -85,B 0,C 180,E1 19035.145,E2 19035.145} C_VEL
LIN {X 0,Y 442.444,Z 683.318,A -85,B 0,C 180,E1 19034.56,E2 19034.56} C_VEL
LIN {X 0,Y 440.519,Z 705.915,A -85,B 0,C 180,E1 19033.762,E2 19033.762} C_VEL
LIN {X 0,Y 438.216,Z 727.136,A -85,B 0,C 180,E1 19032.781,E2 19032.781} C_VEL
LIN {X 0,Y 435.375,Z 749.542,A -85,B 0,C 180,E1 19031.493,E2 19031.493} C_VEL
LIN {X 0,Y 432.605,Z 768.899,A -85,B 0,C 180,E1 19030.151,E2 19030.151} C_VEL
LIN {X 0,Y 429.367,Z 789.589,A -85,B 0,C 180,E1 19028.442,E2 19028.442} C_VEL
LIN {X 0,Y 426.161,Z 809.296,A -85,B 0,C 180,E1 19026.535,E2 19026.535} C_VEL
LIN {X 0,Y 423.022,Z 827.401,A -85,B 0,C 180,E1 19024.475,E2 19024.475} C_VEL
LIN {X 0,Y 419.85,Z 845.986,A -85,B 0,C 180,E1 19022.027,E2 19022.027} C_VEL
LIN {X 0,Y 417.137,Z 862.01,A -85,B 0,C 180,E1 19019.587,E2 19019.587} C_VEL
LIN {X 0,Y 414.651,Z 877.435,A -85,B 0,C 180,E1 19016.85,E2 19016.85} C_VEL
LIN {X 0,Y 412.555,Z 891.441,A -85,B 0,C 180,E1 19013.98,E2 19013.98} C_VEL
LIN {X 0,Y 411.007,Z 902.785,A -85,B 0,C 180,E1 19011.25,E2 19011.25} C_VEL
LIN {X 0,Y 409.743,Z 913.649,A -85,B 0,C 180,E1 19008.199,E2 19008.199} C_VEL
LIN {X 0,Y 408.923,Z 921.759,A -85,B 0,C 180,E1 19005.455,E2 19005.455} C_VEL
LIN {X 0,Y 408.408,Z 928.416,A -85,B 0,C 180,E1 19002.727,E2 19002.727} C_VEL
LIN {X 0,Y 408.084,Z 933.845,A -85,B 0,C 180,E1 18999.589,E2 18999.589} C_VEL
LIN {X 0,Y 407.957,Z 937.44,A -85,B 0,C 180,E1 18996.755,E2 18996.755} C_VEL
LIN {X 0,Y 407.911,Z 939.984,A -85,B 0,C 180,E1 18993.512,E2 18993.512} C_VEL
LIN {X 0,Y 407.904,Z 940.871,A -85,B 0,C 180,E1 18990.841,E2 18990.841} C_VEL
LIN {X 0,Y 407.906,Z 940.595,A -85,B 0,C 180,E1 18987.751,E2 18987.751} C_VEL
LIN {X 0,Y 407.919,Z 938.839,A -85,B 0,C 180,E1 18984.795,E2 18984.795} C_VEL
LIN {X 0,Y 408.002,Z 935.839,A -85,B 0,C 180,E1 18981.827,E2 18981.827} C_VEL
LIN {X 0,Y 408.223,Z 931.079,A -85,B 0,C 180,E1 18978.699,E2 18978.699} C_VEL
LIN {X 0,Y 408.547,Z 926.471,A -85,B 0,C 180,E1 18976.41,E2 18976.41} C_VEL
LIN {X 0,Y 409.233,Z 918.621,A -85,B 0,C 180,E1 18973.388,E2 18973.388} C_VEL
LIN {X 0,Y 410.22,Z 909.312,A -85,B 0,C 180,E1 18970.492,E2 18970.492} C_VEL
LIN {X 0,Y 411.624,Z 898.42,A -85,B 0,C 180,E1 18967.581,E2 18967.581} C_VEL
LIN {X 0,Y 413.438,Z 885.844,A -85,B 0,C 180,E1 18964.753,E2 18964.753} C_VEL
LIN {X 0,Y 415.697,Z 871.638,A -85,B 0,C 180,E1 18961.973,E2 18961.973} C_VEL
LIN {X 0,Y 418.138,Z 857.211,A -85,B 0,C 180,E1 18959.539,E2 18959.539} C_VEL
LIN {X 0,Y 421.291,Z 839.23,A -85,B 0,C 180,E1 18956.907,E2 18956.907} C_VEL
LIN {X 0,Y 424.42,Z 821.818,A -85,B 0,C 180,E1 18954.703,E2 18954.703} C_VEL
LIN {X 0,Y 427.704,Z 802.689,A -85,B 0,C 180,E1 18952.639,E2 18952.639} C_VEL
LIN {X 0,Y 431.137,Z 782.43,A -85,B 0,C 180,E1 18950.768,E2 18950.768} C_VEL
LIN {X 0,Y 434.147,Z 763.166,A -85,B 0,C 180,E1 18949.262,E2 18949.262} C_VEL
LIN {X 0,Y 437.282,Z 740.852,A -85,B 0,C 180,E1 18947.803,E2 18947.803} C_VEL
LIN {X 0,Y 440.048,Z 719.082,A -85,B 0,C 180,E1 18946.643,E2 18946.643} C_VEL
LIN {X 0,Y 442.262,Z 697.217,A -85,B 0,C 180,E1 18945.738,E2 18945.738} C_VEL
LIN {X 0,Y 444.13,Z 674.506,A -85,B 0,C 180,E1 18945.021,E2 18945.021} C_VEL
LIN {X 0,Y 445.262,Z 652.36,A -85,B 0,C 180,E1 18944.534,E2 18944.534} C_VEL
LIN {X 0,Y 450.382,Z 446.048,A -85,B 0,C 180,E1 18940.96,E2 18940.96} C_VEL
LIN {X 0,Y 452.972,Z 344.523,A -85,B 0,C 180,E1 18939.136,E2 18939.136} C_VEL
LIN {X 0,Y 451.153,Z 323.277,A -85,B 0,C 180,E1 18938.437,E2 18938.437} C_VEL
LIN {X 0,Y 451.135,Z 322.188,A -85,B 0,C 180,E1 18938.358,E2 18938.358} C_VEL
LIN {X 0,Y 440.979,Z 302.552,A -85,B 0,C 180,E1 18935.482,E2 18935.482} C_VEL
LIN {X 0,Y 431.655,Z 285.73,A -85,B 0,C 180,E1 18932.664,E2 18932.664} C_VEL
LIN {X 0,Y 424.322,Z 273.177,A -85,B 0,C 180,E1 18930.283,E2 18930.283} C_VEL
LIN {X 0,Y 420.941,Z 267.666,A -85,B 0,C 180,E1 18929.14,E2 18929.14} C_VEL
LIN {X 0,Y 418.429,Z 263.353,A -85,B 0,C 180,E1 18928.238,E2 18928.238} C_VEL
LIN {X 0,Y 415.587,Z 258.625,A -85,B 0,C 180,E1 18927.202,E2 18927.202} C_VEL
LIN {X 0,Y 413.394,Z 255.51,A -85,B 0,C 180,E1 18926.426,E2 18926.426} C_VEL
LIN {X 0,Y 412.512,Z 253.429,A -85,B 0,C 180,E1 18926.022,E2 18926.022} C_VEL
LIN {X 0,Y 410.235,Z 250.763,A -85,B 0,C 180,E1 18925.248,E2 18925.248} C_VEL
LIN {X 0,Y 409.451,Z 248.359,A -85,B 0,C 180,E1 18924.712,E2 18924.712} C_VEL
LIN {X 0,Y 409.387,Z 248.038,A -85,B 0,C 180,E1 18922.961,E2 18922.961} C_VEL
LIN {X 0,Y 409.386,Z 248.035,A -85,B 0,C 180,E1 18919.104,E2 18919.104} C_VEL
LIN {X 0,Y 409.388,Z 248.034,A -85,B 0,C 180,E1 18915.149,E2 18915.149} C_VEL
LIN {X 0,Y 409.397,Z 248.036,A -85,B 0,C 180,E1 18911.267,E2 18911.267} C_VEL
LIN {X 0,Y 409.412,Z 248.046,A -85,B 0,C 180,E1 18907.437,E2 18907.437} C_VEL
LIN {X 0,Y 409.434,Z 248.049,A -85,B 0,C 180,E1 18903.641,E2 18903.641} C_VEL
LIN {X 0,Y 409.448,Z 248.031,A -85,B 0,C 180,E1 18899.721,E2 18899.721} C_VEL
LIN {X 0,Y 409.435,Z 248.022,A -85,B 0,C 180,E1 18895.799,E2 18895.799} C_VEL
LIN {X 0,Y 409.427,Z 248.025,A -85,B 0,C 180,E1 18891.999,E2 18891.999} C_VEL
LIN {X 0,Y 409.418,Z 248.049,A -85,B 0,C 180,E1 18888.163,E2 18888.163} C_VEL
LIN {X 0,Y 409.416,Z 248.042,A -85,B 0,C 180,E1 18884.272,E2 18884.272} C_VEL
LIN {X 0,Y 409.416,Z 248.021,A -85,B 0,C 180,E1 18880.305,E2 18880.305} C_VEL
LIN {X 0,Y 409.421,Z 248.028,A -85,B 0,C 180,E1 18876.391,E2 18876.391} C_VEL
LIN {X 0,Y 409.432,Z 248.046,A -85,B 0,C 180,E1 18872.435,E2 18872.435} C_VEL
LIN {X 0,Y 409.436,Z 248.044,A -85,B 0,C 180,E1 18868.494,E2 18868.494} C_VEL
LIN {X 0,Y 409.435,Z 248.025,A -85,B 0,C 180,E1 18864.637,E2 18864.637} C_VEL
LIN {X 0,Y 409.435,Z 248.021,A -85,B 0,C 180,E1 18860.727,E2 18860.727} C_VEL
LIN {X 0,Y 409.435,Z 248.032,A -85,B 0,C 180,E1 18856.862,E2 18856.862} C_VEL
LIN {X 0,Y 409.433,Z 248.041,A -85,B 0,C 180,E1 18852.895,E2 18852.895} C_VEL
LIN {X 0,Y 409.444,Z 248.045,A -85,B 0,C 180,E1 18849.054,E2 18849.054} C_VEL
LIN {X 0,Y 409.437,Z 248.047,A -85,B 0,C 180,E1 18845.022,E2 18845.022} C_VEL
LIN {X 0,Y 409.441,Z 248.04,A -85,B 0,C 180,E1 18841.004,E2 18841.004} C_VEL
LIN {X 0,Y 409.466,Z 248.307,A -85,B 0,C 180,E1 18838.177,E2 18838.177} C_VEL
LIN {X 0,Y 410.938,Z 251.79,A -85,B 0,C 180,E1 18837.368,E2 18837.368} C_VEL
LIN {X 0,Y 412.517,Z 253.884,A -85,B 0,C 180,E1 18836.798,E2 18836.798} C_VEL
LIN {X 0,Y 414.668,Z 257.747,A -85,B 0,C 180,E1 18835.924,E2 18835.924} C_VEL
LIN {X 0,Y 418.939,Z 265.405,A -85,B 0,C 180,E1 18834.261,E2 18834.261} C_VEL
LIN {X 0,Y 423.444,Z 273.452,A -85,B 0,C 180,E1 18832.597,E2 18832.597} C_VEL
LIN {X 0,Y 431.023,Z 288.168,A -85,B 0,C 180,E1 18829.868,E2 18829.868} C_VEL
LIN {X 0,Y 438.616,Z 304.143,A -85,B 0,C 180,E1 18827.23,E2 18827.23} C_VEL
LIN {X 0,Y 443.073,Z 314.544,A -85,B 0,C 180,E1 18825.679,E2 18825.679} C_VEL
LIN {X 0,Y 437.062,Z 369.257,A -85,B 0,C 180,E1 18821.615,E2 18821.615} C_VEL
LIN {X 0,Y 433.816,Z 402.621,A -85,B 0,C 180,E1 18819.19,E2 18819.19} C_VEL
LIN {X 0,Y 438.159,Z 444.967,A -85,B 0,C 180,E1 18817.744,E2 18817.744} C_VEL
LIN {X 0,Y 438.034,Z 448.519,A -85,B 0,C 180,E1 18817.679,E2 18817.679} C_VEL
LIN {X 0,Y 436.997,Z 456.205,A -85,B 0,C 180,E1 18817.624,E2 18817.624} C_VEL
LIN {X 0,Y 431.478,Z 476.691,A -85,B 0,C 180,E1 18817.779,E2 18817.779} C_VEL
LIN {X 0,Y 430.67,Z 483.285,A -85,B 0,C 180,E1 18817.718,E2 18817.718} C_VEL
LIN {X 0,Y 425.179,Z 633.116,A -85,B 0,C 180,E1 18814.849,E2 18814.849} C_VEL
LIN {X 0,Y 423.797,Z 653.567,A -85,B 0,C 180,E1 18814.218,E2 18814.218} C_VEL
LIN {X 0,Y 422.129,Z 672.244,A -85,B 0,C 180,E1 18813.396,E2 18813.396} C_VEL
LIN {X 0,Y 420.077,Z 690.845,A -85,B 0,C 180,E1 18812.32,E2 18812.32} C_VEL
LIN {X 0,Y 417.671,Z 709.304,A -85,B 0,C 180,E1 18810.962,E2 18810.962} C_VEL
LIN {X 0,Y 415.133,Z 726.545,A -85,B 0,C 180,E1 18809.38,E2 18809.38} C_VEL
LIN {X 0,Y 412.664,Z 742.094,A -85,B 0,C 180,E1 18807.641,E2 18807.641} C_VEL
LIN {X 0,Y 410.231,Z 756.648,A -85,B 0,C 180,E1 18805.668,E2 18805.668} C_VEL
LIN {X 0,Y 407.986,Z 769.716,A -85,B 0,C 180,E1 18803.529,E2 18803.529} C_VEL
LIN {X 0,Y 406.02,Z 781.343,A -85,B 0,C 180,E1 18801.219,E2 18801.219} C_VEL
LIN {X 0,Y 404.358,Z 791.532,A -85,B 0,C 180,E1 18798.737,E2 18798.737} C_VEL
LIN {X 0,Y 403.109,Z 799.814,A -85,B 0,C 180,E1 18796.226,E2 18796.226} C_VEL
LIN {X 0,Y 402.198,Z 806.707,A -85,B 0,C 180,E1 18793.538,E2 18793.538} C_VEL
LIN {X 0,Y 401.606,Z 811.85,A -85,B 0,C 180,E1 18790.816,E2 18790.816} C_VEL
LIN {X 0,Y 401.293,Z 815.309,A -85,B 0,C 180,E1 18788.055,E2 18788.055} C_VEL
LIN {X 0,Y 401.164,Z 817.113,A -85,B 0,C 180,E1 18785.248,E2 18785.248} C_VEL
LIN {X 0,Y 401.195,Z 817.267,A -85,B 0,C 180,E1 18782.524,E2 18782.524} C_VEL
LIN {X 0,Y 401.382,Z 815.808,A -85,B 0,C 180,E1 18779.791,E2 18779.791} C_VEL
LIN {X 0,Y 401.783,Z 812.601,A -85,B 0,C 180,E1 18776.978,E2 18776.978} C_VEL
LIN {X 0,Y 402.519,Z 807.455,A -85,B 0,C 180,E1 18774.113,E2 18774.113} C_VEL
LIN {X 0,Y 403.584,Z 800.613,A -85,B 0,C 180,E1 18771.37,E2 18771.37} C_VEL
LIN {X 0,Y 405.05,Z 792.193,A -85,B 0,C 180,E1 18768.772,E2 18768.772} C_VEL
LIN {X 0,Y 406.87,Z 782.299,A -85,B 0,C 180,E1 18766.33,E2 18766.33} C_VEL
LIN {X 0,Y 409.109,Z 770.448,A -85,B 0,C 180,E1 18763.954,E2 18763.954} C_VEL
LIN {X 0,Y 411.617,Z 757.233,A -85,B 0,C 180,E1 18761.781,E2 18761.781} C_VEL
LIN {X 0,Y 414.199,Z 743.145,A -85,B 0,C 180,E1 18759.861,E2 18759.861} C_VEL
LIN {X 0,Y 416.867,Z 727.756,A -85,B 0,C 180,E1 18758.124,E2 18758.124} C_VEL
LIN {X 0,Y 419.589,Z 710.871,A -85,B 0,C 180,E1 18756.564,E2 18756.564} C_VEL
LIN {X 0,Y 422.159,Z 692.712,A -85,B 0,C 180,E1 18755.207,E2 18755.207} C_VEL
LIN {X 0,Y 424.463,Z 673.864,A -85,B 0,C 180,E1 18754.098,E2 18754.098} C_VEL
LIN {X 0,Y 426.394,Z 654.264,A -85,B 0,C 180,E1 18753.224,E2 18753.224} C_VEL
LIN {X 0,Y 427.902,Z 634.185,A -85,B 0,C 180,E1 18752.594,E2 18752.594} C_VEL
LIN {X 0,Y 434.305,Z 492.173,A -85,B 0,C 180,E1 18749.752,E2 18749.752} C_VEL
LIN {X 0,Y 436.252,Z 445.351,A -85,B 0,C 180,E1 18748.826,E2 18748.826} C_VEL
LIN {X 0,Y 431.417,Z 394.717,A -85,B 0,C 180,E1 18746.843,E2 18746.843} C_VEL
LIN {X 0,Y 438.089,Z 341.865,A -85,B 0,C 180,E1 18742.829,E2 18742.829} C_VEL
LIN {X 0,Y 440.712,Z 322.649,A -85,B 0,C 180,E1 18741.353,E2 18741.353} C_VEL
LIN {X 0,Y 433.903,Z 307.3,A -85,B 0,C 180,E1 18738.681,E2 18738.681} C_VEL
LIN {X 0,Y 427.501,Z 293.934,A -85,B 0,C 180,E1 18736.02,E2 18736.02} C_VEL
LIN {X 0,Y 420.526,Z 280.721,A -85,B 0,C 180,E1 18732.914,E2 18732.914} C_VEL
LIN {X 0,Y 417.156,Z 275.061,A -85,B 0,C 180,E1 18731.334,E2 18731.334} C_VEL
LIN {X 0,Y 414.566,Z 270.499,A -85,B 0,C 180,E1 18730,E2 18730} C_VEL
LIN {X 0,Y 412.358,Z 266.715,A -85,B 0,C 180,E1 18728.786,E2 18728.786} C_VEL
LIN {X 0,Y 411.353,Z 265.22,A -85,B 0,C 180,E1 18728.245,E2 18728.245} C_VEL
LIN {X 0,Y 409.241,Z 261.866,A -85,B 0,C 180,E1 18727.016,E2 18727.016} C_VEL
LIN {X 0,Y 408.465,Z 260.264,A -85,B 0,C 180,E1 18726.465,E2 18726.465} C_VEL
LIN {X 0,Y 405.98,Z 257.051,A -85,B 0,C 180,E1 18724.944,E2 18724.944} C_VEL
LIN {X 0,Y 404.951,Z 254.743,A -85,B 0,C 180,E1 18724.074,E2 18724.074} C_VEL
LIN {X 0,Y 402.192,Z 251.557,A -85,B 0,C 180,E1 18722.078,E2 18722.078} C_VEL
LIN {X 0,Y 401.487,Z 249.367,A -85,B 0,C 180,E1 18720.998,E2 18720.998} C_VEL
LIN {X 0,Y 401.469,Z 249.035,A -85,B 0,C 180,E1 18718.572,E2 18718.572} C_VEL
LIN {X 0,Y 401.457,Z 249.032,A -85,B 0,C 180,E1 18714.569,E2 18714.569} C_VEL
LIN {X 0,Y 401.432,Z 249.031,A -85,B 0,C 180,E1 18710.827,E2 18710.827} C_VEL
LIN {X 0,Y 401.424,Z 249.037,A -85,B 0,C 180,E1 18707.045,E2 18707.045} C_VEL
LIN {X 0,Y 401.422,Z 249.039,A -85,B 0,C 180,E1 18703.024,E2 18703.024} C_VEL
LIN {X 0,Y 401.494,Z 249.32,A -85,B 0,C 180,E1 18701.712,E2 18701.712} C_VEL
LIN {X 0,Y 402.972,Z 252.791,A -85,B 0,C 180,E1 18699.976,E2 18699.976} C_VEL
LIN {X 0,Y 405.581,Z 255.52,A -85,B 0,C 180,E1 18698.297,E2 18698.297} C_VEL
LIN {X 0,Y 407.389,Z 259.148,A -85,B 0,C 180,E1 18696.974,E2 18696.974} C_VEL
LIN {X 0,Y 409.27,Z 261.006,A -85,B 0,C 180,E1 18696.016,E2 18696.016} C_VEL
LIN {X 0,Y 411.211,Z 264.827,A -85,B 0,C 180,E1 18694.817,E2 18694.817} C_VEL
LIN {X 0,Y 412.726,Z 266.388,A -85,B 0,C 180,E1 18694.147,E2 18694.147} C_VEL
LIN {X 0,Y 415.063,Z 270.665,A -85,B 0,C 180,E1 18692.916,E2 18692.916} C_VEL
LIN {X 0,Y 416.266,Z 272.399,A -85,B 0,C 180,E1 18692.381,E2 18692.381} C_VEL
LIN {X 0,Y 419.844,Z 278.463,A -85,B 0,C 180,E1 18690.777,E2 18690.777} C_VEL
LIN {X 0,Y 424.425,Z 286.01,A -85,B 0,C 180,E1 18688.941,E2 18688.941} C_VEL
LIN {X 0,Y 431.662,Z 299.378,A -85,B 0,C 180,E1 18686.226,E2 18686.226} C_VEL
LIN {X 0,Y 439.11,Z 314.194,A -85,B 0,C 180,E1 18683.699,E2 18683.699} C_VEL
LIN {X 0,Y 444.221,Z 325.507,A -85,B 0,C 180,E1 18682.044,E2 18682.044} C_VEL
LIN {X 0,Y 443.975,Z 330.231,A -85,B 0,C 180,E1 18681.795,E2 18681.795} C_VEL
LIN {X 0,Y 445.387,Z 348.554,A -85,B 0,C 180,E1 18681.222,E2 18681.222} C_VEL
LIN {X 0,Y 440.319,Z 547.12,A -85,B 0,C 180,E1 18677.73,E2 18677.73} C_VEL
LIN {X 0,Y 437.651,Z 660.216,A -85,B 0,C 180,E1 18675.791,E2 18675.791} C_VEL
LIN {X 0,Y 436.097,Z 682.954,A -85,B 0,C 180,E1 18675.206,E2 18675.206} C_VEL
LIN {X 0,Y 434.064,Z 705.592,A -85,B 0,C 180,E1 18674.399,E2 18674.399} C_VEL
LIN {X 0,Y 431.633,Z 726.937,A -85,B 0,C 180,E1 18673.4,E2 18673.4} C_VEL
LIN {X 0,Y 428.688,Z 749.1,A -85,B 0,C 180,E1 18672.108,E2 18672.108} C_VEL
LIN {X 0,Y 425.793,Z 768.431,A -85,B 0,C 180,E1 18670.751,E2 18670.751} C_VEL
LIN {X 0,Y 422.395,Z 789.033,A -85,B 0,C 180,E1 18669.022,E2 18669.022} C_VEL
LIN {X 0,Y 419.075,Z 808.332,A -85,B 0,C 180,E1 18667.128,E2 18667.128} C_VEL
LIN {X 0,Y 415.739,Z 826.747,A -85,B 0,C 180,E1 18664.999,E2 18664.999} C_VEL
LIN {X 0,Y 412.311,Z 845.723,A -85,B 0,C 180,E1 18662.445,E2 18662.445} C_VEL
LIN {X 0,Y 409.398,Z 862.177,A -85,B 0,C 180,E1 18659.88,E2 18659.88} C_VEL
LIN {X 0,Y 406.888,Z 876.945,A -85,B 0,C 180,E1 18657.183,E2 18657.183} C_VEL
LIN {X 0,Y 404.672,Z 891.032,A -85,B 0,C 180,E1 18654.212,E2 18654.212} C_VEL
LIN {X 0,Y 403.054,Z 902.475,A -85,B 0,C 180,E1 18651.385,E2 18651.385} C_VEL
LIN {X 0,Y 401.718,Z 913.618,A -85,B 0,C 180,E1 18648.125,E2 18648.125} C_VEL
LIN {X 0,Y 400.91,Z 921.587,A -85,B 0,C 180,E1 18645.327,E2 18645.327} C_VEL
LIN {X 0,Y 400.353,Z 929.004,A -85,B 0,C 180,E1 18642.108,E2 18642.108} C_VEL
LIN {X 0,Y 400.069,Z 933.939,A -85,B 0,C 180,E1 18639.347,E2 18639.347} C_VEL
LIN {X 0,Y 399.946,Z 937.922,A -85,B 0,C 180,E1 18636.314,E2 18636.314} C_VEL
LIN {X 0,Y 399.911,Z 940.109,A -85,B 0,C 180,E1 18633.295,E2 18633.295} C_VEL
LIN {X 0,Y 399.9,Z 940.938,A -85,B 0,C 180,E1 18630.428,E2 18630.428} C_VEL
LIN {X 0,Y 399.911,Z 940.384,A -85,B 0,C 180,E1 18627.276,E2 18627.276} C_VEL
LIN {X 0,Y 399.92,Z 938.653,A -85,B 0,C 180,E1 18624.547,E2 18624.547} C_VEL
LIN {X 0,Y 400.004,Z 935.661,A -85,B 0,C 180,E1 18621.807,E2 18621.807} C_VEL
LIN {X 0,Y 400.247,Z 930.444,A -85,B 0,C 180,E1 18618.617,E2 18618.617} C_VEL
LIN {X 0,Y 400.678,Z 924.548,A -85,B 0,C 180,E1 18615.843,E2 18615.843} C_VEL
LIN {X 0,Y 401.515,Z 915.545,A -85,B 0,C 180,E1 18612.462,E2 18612.462} C_VEL
LIN {X 0,Y 402.566,Z 906.484,A -85,B 0,C 180,E1 18609.651,E2 18609.651} C_VEL
LIN {X 0,Y 404.207,Z 894.548,A -85,B 0,C 180,E1 18606.53,E2 18606.53} C_VEL
LIN {X 0,Y 406.189,Z 881.946,A -85,B 0,C 180,E1 18603.698,E2 18603.698} C_VEL
LIN {X 0,Y 408.568,Z 867.976,A -85,B 0,C 180,E1 18601.016,E2 18601.016} C_VEL
LIN {X 0,Y 411.372,Z 852.517,A -85,B 0,C 180,E1 18598.412,E2 18598.412} C_VEL
LIN {X 0,Y 414.529,Z 835.54,A -85,B 0,C 180,E1 18595.971,E2 18595.971} C_VEL
LIN {X 0,Y 418.156,Z 816.03,A -85,B 0,C 180,E1 18593.556,E2 18593.556} C_VEL
LIN {X 0,Y 421.59,Z 797.423,A -85,B 0,C 180,E1 18591.583,E2 18591.583} C_VEL
LIN {X 0,Y 424.89,Z 778.167,A -85,B 0,C 180,E1 18589.849,E2 18589.849} C_VEL
LIN {X 0,Y 428.215,Z 757.76,A -85,B 0,C 180,E1 18588.281,E2 18588.281} C_VEL
LIN {X 0,Y 431.105,Z 737.617,A -85,B 0,C 180,E1 18587.009,E2 18587.009} C_VEL
LIN {X 0,Y 433.948,Z 715.418,A -85,B 0,C 180,E1 18585.859,E2 18585.859} C_VEL
LIN {X 0,Y 436.107,Z 694.694,A -85,B 0,C 180,E1 18585.012,E2 18585.012} C_VEL
LIN {X 0,Y 438.025,Z 671.084,A -85,B 0,C 180,E1 18584.294,E2 18584.294} C_VEL
LIN {X 0,Y 439.164,Z 648.003,A -85,B 0,C 180,E1 18583.802,E2 18583.802} C_VEL
LIN {X 0,Y 444.422,Z 444.937,A -85,B 0,C 180,E1 18580.257,E2 18580.257} C_VEL
LIN {X 0,Y 447.114,Z 345.891,A -85,B 0,C 180,E1 18578.46,E2 18578.46} C_VEL
LIN {X 0,Y 445.209,Z 326.104,A -85,B 0,C 180,E1 18577.794,E2 18577.794} C_VEL
LIN {X 0,Y 442.847,Z 321.819,A -85,B 0,C 180,E1 18577.235,E2 18577.235} C_VEL
LIN {X 0,Y 433.731,Z 304.359,A -85,B 0,C 180,E1 18574.548,E2 18574.548} C_VEL
LIN {X 0,Y 425.016,Z 288.598,A -85,B 0,C 180,E1 18571.801,E2 18571.801} C_VEL
LIN {X 0,Y 418.506,Z 277.601,A -85,B 0,C 180,E1 18569.64,E2 18569.64} C_VEL
LIN {X 0,Y 413.408,Z 269.052,A -85,B 0,C 180,E1 18567.826,E2 18567.826} C_VEL
LIN {X 0,Y 410.568,Z 264.445,A -85,B 0,C 180,E1 18566.778,E2 18566.778} C_VEL
LIN {X 0,Y 408.238,Z 260.313,A -85,B 0,C 180,E1 18565.847,E2 18565.847} C_VEL
LIN {X 0,Y 405.399,Z 256.306,A -85,B 0,C 180,E1 18564.789,E2 18564.789} C_VEL
LIN {X 0,Y 404.537,Z 254.385,A -85,B 0,C 180,E1 18564.379,E2 18564.379} C_VEL
LIN {X 0,Y 402.345,Z 251.842,A -85,B 0,C 180,E1 18563.585,E2 18563.585} C_VEL
LIN {X 0,Y 401.5,Z 249.386,A -85,B 0,C 180,E1 18563.016,E2 18563.016} C_VEL
LIN {X 0,Y 401.475,Z 249.018,A -85,B 0,C 180,E1 18561.936,E2 18561.936} C_VEL
LIN {X 0,Y 401.491,Z 249.015,A -85,B 0,C 180,E1 18558.138,E2 18558.138} C_VEL
LIN {X 0,Y 401.503,Z 249.013,A -85,B 0,C 180,E1 18554.126,E2 18554.126} C_VEL
LIN {X 0,Y 401.487,Z 249.013,A -85,B 0,C 180,E1 18550.185,E2 18550.185} C_VEL
LIN {X 0,Y 401.469,Z 249.017,A -85,B 0,C 180,E1 18546.423,E2 18546.423} C_VEL
LIN {X 0,Y 401.465,Z 249.029,A -85,B 0,C 180,E1 18542.57,E2 18542.57} C_VEL
LIN {X 0,Y 401.465,Z 249.039,A -85,B 0,C 180,E1 18538.716,E2 18538.716} C_VEL
LIN {X 0,Y 401.467,Z 249.028,A -85,B 0,C 180,E1 18534.713,E2 18534.713} C_VEL
LIN {X 0,Y 401.473,Z 249.01,A -85,B 0,C 180,E1 18530.829,E2 18530.829} C_VEL
LIN {X 0,Y 401.486,Z 249.016,A -85,B 0,C 180,E1 18526.902,E2 18526.902} C_VEL
LIN {X 0,Y 401.497,Z 249.034,A -85,B 0,C 180,E1 18522.999,E2 18522.999} C_VEL
LIN {X 0,Y 401.503,Z 249.027,A -85,B 0,C 180,E1 18518.986,E2 18518.986} C_VEL
LIN {X 0,Y 401.5,Z 249.01,A -85,B 0,C 180,E1 18515.024,E2 18515.024} C_VEL
LIN {X 0,Y 401.501,Z 249.01,A -85,B 0,C 180,E1 18511.112,E2 18511.112} C_VEL
LIN {X 0,Y 401.5,Z 249.03,A -85,B 0,C 180,E1 18507.121,E2 18507.121} C_VEL
LIN {X 0,Y 401.5,Z 249.037,A -85,B 0,C 180,E1 18503.073,E2 18503.073} C_VEL
LIN {X 0,Y 401.5,Z 249.022,A -85,B 0,C 180,E1 18499.085,E2 18499.085} C_VEL
LIN {X 0,Y 401.495,Z 249.013,A -85,B 0,C 180,E1 18495.191,E2 18495.191} C_VEL
LIN {X 0,Y 401.503,Z 249.011,A -85,B 0,C 180,E1 18491.232,E2 18491.232} C_VEL
LIN {X 0,Y 401.495,Z 249.014,A -85,B 0,C 180,E1 18487.401,E2 18487.401} C_VEL
LIN {X 0,Y 401.499,Z 249.014,A -85,B 0,C 180,E1 18483.463,E2 18483.463} C_VEL
LIN {X 0,Y 401.539,Z 249.273,A -85,B 0,C 180,E1 18479.788,E2 18479.788} C_VEL
LIN {X 0,Y 403.11,Z 252.928,A -85,B 0,C 180,E1 18478.89,E2 18478.89} C_VEL
LIN {X 0,Y 404.638,Z 254.819,A -85,B 0,C 180,E1 18478.324,E2 18478.324} C_VEL
LIN {X 0,Y 406.661,Z 258.62,A -85,B 0,C 180,E1 18477.43,E2 18477.43} C_VEL
LIN {X 0,Y 407.791,Z 260.466,A -85,B 0,C 180,E1 18476.976,E2 18476.976} C_VEL
LIN {X 0,Y 410.764,Z 265.728,A -85,B 0,C 180,E1 18475.761,E2 18475.761} C_VEL
LIN {X 0,Y 415.763,Z 274.55,A -85,B 0,C 180,E1 18473.831,E2 18473.831} C_VEL
LIN {X 0,Y 422.73,Z 287.85,A -85,B 0,C 180,E1 18471.217,E2 18471.217} C_VEL
LIN {X 0,Y 430.056,Z 302.889,A -85,B 0,C 180,E1 18468.575,E2 18468.575} C_VEL
LIN {X 0,Y 436.797,Z 318.133,A -85,B 0,C 180,E1 18466.184,E2 18466.184} C_VEL
LIN {X 0,Y 430.494,Z 372.985,A -85,B 0,C 180,E1 18462.067,E2 18462.067} C_VEL
LIN {X 0,Y 427.562,Z 401.728,A -85,B 0,C 180,E1 18459.958,E2 18459.958} C_VEL
LIN {X 0,Y 432.018,Z 446.086,A -85,B 0,C 180,E1 18458.408,E2 18458.408} C_VEL
LIN {X 0,Y 430.67,Z 483.285,A -85,B 0,C 180,E1 18457.718,E2 18457.718} C_VEL
LIN {X 0,Y 429.634,Z 490.968,A -85,B 0,C 180,E1 18457.659,E2 18457.659} C_VEL
LIN {X 0,Y 424.078,Z 511.448,A -85,B 0,C 180,E1 18457.81,E2 18457.81} C_VEL
LIN {X 0,Y 423.244,Z 518.042,A -85,B 0,C 180,E1 18457.751,E2 18457.751} C_VEL
LIN {X 0,Y 418.711,Z 634.249,A -85,B 0,C 180,E1 18455.475,E2 18455.475} C_VEL
LIN {X 0,Y 417.252,Z 654.544,A -85,B 0,C 180,E1 18454.831,E2 18454.831} C_VEL
LIN {X 0,Y 415.518,Z 673.053,A -85,B 0,C 180,E1 18454.003,E2 18454.003} C_VEL
LIN {X 0,Y 413.369,Z 691.613,A -85,B 0,C 180,E1 18452.913,E2 18452.913} C_VEL
LIN {X 0,Y 410.844,Z 710.06,A -85,B 0,C 180,E1 18451.535,E2 18451.535} C_VEL
LIN {X 0,Y 408.288,Z 726.66,A -85,B 0,C 180,E1 18450.001,E2 18450.001} C_VEL
LIN {X 0,Y 405.572,Z 742.895,A -85,B 0,C 180,E1 18448.165,E2 18448.165} C_VEL
LIN {X 0,Y 403,Z 757.482,A -85,B 0,C 180,E1 18446.161,E2 18446.161} C_VEL
LIN {X 0,Y 400.616,Z 770.589,A -85,B 0,C 180,E1 18443.985,E2 18443.985} C_VEL
LIN {X 0,Y 398.52,Z 782.255,A -85,B 0,C 180,E1 18441.634,E2 18441.634} C_VEL
LIN {X 0,Y 396.742,Z 792.486,A -85,B 0,C 180,E1 18439.106,E2 18439.106} C_VEL
LIN {X 0,Y 395.395,Z 800.814,A -85,B 0,C 180,E1 18436.549,E2 18436.549} C_VEL
LIN {X 0,Y 394.405,Z 807.752,A -85,B 0,C 180,E1 18433.81,E2 18433.81} C_VEL
LIN {X 0,Y 393.754,Z 812.944,A -85,B 0,C 180,E1 18431.034,E2 18431.034} C_VEL
LIN {X 0,Y 393.407,Z 816.456,A -85,B 0,C 180,E1 18428.221,E2 18428.221} C_VEL
LIN {X 0,Y 393.264,Z 818.319,A -85,B 0,C 180,E1 18425.359,E2 18425.359} C_VEL
LIN {X 0,Y 393.295,Z 818.488,A -85,B 0,C 180,E1 18422.441,E2 18422.441} C_VEL
LIN {X 0,Y 393.504,Z 817.006,A -85,B 0,C 180,E1 18419.628,E2 18419.628} C_VEL
LIN {X 0,Y 393.949,Z 813.774,A -85,B 0,C 180,E1 18416.758,E2 18416.758} C_VEL
LIN {X 0,Y 394.733,Z 808.749,A -85,B 0,C 180,E1 18413.902,E2 18413.902} C_VEL
LIN {X 0,Y 395.9,Z 801.813,A -85,B 0,C 180,E1 18411.064,E2 18411.064} C_VEL
LIN {X 0,Y 397.494,Z 793.308,A -85,B 0,C 180,E1 18408.392,E2 18408.392} C_VEL
LIN {X 0,Y 399.494,Z 783.136,A -85,B 0,C 180,E1 18405.844,E2 18405.844} C_VEL
LIN {X 0,Y 401.813,Z 771.661,A -85,B 0,C 180,E1 18403.504,E2 18403.504} C_VEL
LIN {X 0,Y 404.483,Z 758.402,A -85,B 0,C 180,E1 18401.285,E2 18401.285} C_VEL
LIN {X 0,Y 407.267,Z 744.06,A -85,B 0,C 180,E1 18399.3,E2 18399.3} C_VEL
LIN {X 0,Y 410.147,Z 728.308,A -85,B 0,C 180,E1 18397.5,E2 18397.5} C_VEL
LIN {X 0,Y 413.01,Z 711.463,A -85,B 0,C 180,E1 18395.928,E2 18395.928} C_VEL
LIN {X 0,Y 415.643,Z 693.825,A -85,B 0,C 180,E1 18394.59,E2 18394.59} C_VEL
LIN {X 0,Y 418.038,Z 675.283,A -85,B 0,C 180,E1 18393.478,E2 18393.478} C_VEL
LIN {X 0,Y 420.117,Z 655.295,A -85,B 0,C 180,E1 18392.566,E2 18392.566} C_VEL
LIN {X 0,Y 421.734,Z 634.942,A -85,B 0,C 180,E1 18391.914,E2 18391.914} C_VEL
LIN {X 0,Y 428.191,Z 499.171,A -85,B 0,C 180,E1 18389.153,E2 18389.153} C_VEL
LIN {X 0,Y 430.504,Z 446.681,A -85,B 0,C 180,E1 18388.106,E2 18388.106} C_VEL
LIN {X 0,Y 425.629,Z 394.227,A -85,B 0,C 180,E1 18386.016,E2 18386.016} C_VEL
LIN {X 0,Y 432.493,Z 342.177,A -85,B 0,C 180,E1 18382.026,E2 18382.026} C_VEL
LIN {X 0,Y 434.715,Z 326.616,A -85,B 0,C 180,E1 18380.815,E2 18380.815} C_VEL
LIN {X 0,Y 427.769,Z 310.777,A -85,B 0,C 180,E1 18377.97,E2 18377.97} C_VEL
LIN {X 0,Y 421.768,Z 298.449,A -85,B 0,C 180,E1 18375.397,E2 18375.397} C_VEL
LIN {X 0,Y 415.871,Z 286.943,A -85,B 0,C 180,E1 18372.637,E2 18372.637} C_VEL
LIN {X 0,Y 412.514,Z 281.206,A -85,B 0,C 180,E1 18371.005,E2 18371.005} C_VEL
LIN {X 0,Y 410.338,Z 277.168,A -85,B 0,C 180,E1 18369.82,E2 18369.82} C_VEL
LIN {X 0,Y 407.859,Z 272.69,A -85,B 0,C 180,E1 18368.387,E2 18368.387} C_VEL
LIN {X 0,Y 405.124,Z 268.594,A -85,B 0,C 180,E1 18366.803,E2 18366.803} C_VEL
LIN {X 0,Y 404.309,Z 266.999,A -85,B 0,C 180,E1 18366.222,E2 18366.222} C_VEL
LIN {X 0,Y 401.948,Z 263.759,A -85,B 0,C 180,E1 18364.708,E2 18364.708} C_VEL
LIN {X 0,Y 401.239,Z 261.812,A -85,B 0,C 180,E1 18364,E2 18364} C_VEL
LIN {X 0,Y 398.514,Z 258.707,A -85,B 0,C 180,E1 18362.012,E2 18362.012} C_VEL
LIN {X 0,Y 397.288,Z 255.887,A -85,B 0,C 180,E1 18360.576,E2 18360.576} C_VEL
LIN {X 0,Y 394.003,Z 251.941,A -85,B 0,C 180,E1 18356.653,E2 18356.653} C_VEL
LIN {X 0,Y 393.551,Z 250.274,A -85,B 0,C 180,E1 18354.606,E2 18354.606} C_VEL
LIN {X 0,Y 393.498,Z 250.038,A -85,B 0,C 180,E1 18350.788,E2 18350.788} C_VEL
LIN {X 0,Y 393.568,Z 250.508,A -85,B 0,C 180,E1 18347.529,E2 18347.529} C_VEL
LIN {X 0,Y 395.429,Z 254.292,A -85,B 0,C 180,E1 18343.85,E2 18343.85} C_VEL
LIN {X 0,Y 397.824,Z 256.585,A -85,B 0,C 180,E1 18341.689,E2 18341.689} C_VEL
LIN {X 0,Y 399.767,Z 260.395,A -85,B 0,C 180,E1 18339.809,E2 18339.809} C_VEL
LIN {X 0,Y 401.762,Z 262.351,A -85,B 0,C 180,E1 18338.541,E2 18338.541} C_VEL
LIN {X 0,Y 403.661,Z 266.158,A -85,B 0,C 180,E1 18337.115,E2 18337.115} C_VEL
LIN {X 0,Y 405.432,Z 268.235,A -85,B 0,C 180,E1 18336.143,E2 18336.143} C_VEL
LIN {X 0,Y 407.834,Z 272.292,A -85,B 0,C 180,E1 18334.749,E2 18334.749} C_VEL
LIN {X 0,Y 408.921,Z 273.88,A -85,B 0,C 180,E1 18334.2,E2 18334.2} C_VEL
LIN {X 0,Y 412.209,Z 279.32,A -85,B 0,C 180,E1 18332.557,E2 18332.557} C_VEL
LIN {X 0,Y 415.442,Z 284.797,A -85,B 0,C 180,E1 18331.069,E2 18331.069} C_VEL
LIN {X 0,Y 420.221,Z 293.015,A -85,B 0,C 180,E1 18329.073,E2 18329.073} C_VEL
LIN {X 0,Y 426.702,Z 305.043,A -85,B 0,C 180,E1 18326.588,E2 18326.588} C_VEL
LIN {X 0,Y 433.997,Z 319.841,A -85,B 0,C 180,E1 18324.021,E2 18324.021} C_VEL
LIN {X 0,Y 438.22,Z 329.416,A -85,B 0,C 180,E1 18322.596,E2 18322.596} C_VEL
LIN {X 0,Y 439.617,Z 349.897,A -85,B 0,C 180,E1 18321.925,E2 18321.925} C_VEL
LIN {X 0,Y 434.257,Z 546.831,A -85,B 0,C 180,E1 18318.422,E2 18318.422} C_VEL
LIN {X 0,Y 431.415,Z 660.118,A -85,B 0,C 180,E1 18316.456,E2 18316.456} C_VEL
LIN {X 0,Y 429.789,Z 682.919,A -85,B 0,C 180,E1 18315.862,E2 18315.862} C_VEL
LIN {X 0,Y 427.674,Z 705.321,A -85,B 0,C 180,E1 18315.054,E2 18315.054} C_VEL
LIN {X 0,Y 425.256,Z 725.584,A -85,B 0,C 180,E1 18314.101,E2 18314.101} C_VEL
LIN {X 0,Y 422.213,Z 747.602,A -85,B 0,C 180,E1 18312.814,E2 18312.814} C_VEL
LIN {X 0,Y 419.029,Z 767.964,A -85,B 0,C 180,E1 18311.371,E2 18311.371} C_VEL
LIN {X 0,Y 415.52,Z 788.241,A -85,B 0,C 180,E1 18309.645,E2 18309.645} C_VEL
LIN {X 0,Y 411.969,Z 807.739,A -85,B 0,C 180,E1 18307.701,E2 18307.701} C_VEL
LIN {X 0,Y 408.519,Z 825.952,A -85,B 0,C 180,E1 18305.559,E2 18305.559} C_VEL
LIN {X 0,Y 404.929,Z 844.753,A -85,B 0,C 180,E1 18302.986,E2 18302.986} C_VEL
LIN {X 0,Y 402.001,Z 860.524,A -85,B 0,C 180,E1 18300.488,E2 18300.488} C_VEL
LIN {X 0,Y 399.332,Z 875.31,A -85,B 0,C 180,E1 18297.754,E2 18297.754} C_VEL
LIN {X 0,Y 397.073,Z 888.908,A -85,B 0,C 180,E1 18294.865,E2 18294.865} C_VEL
LIN {X 0,Y 395.339,Z 900.459,A -85,B 0,C 180,E1 18291.98,E2 18291.98} C_VEL
LIN {X 0,Y 393.927,Z 911.385,A -85,B 0,C 180,E1 18288.783,E2 18288.783} C_VEL
LIN {X 0,Y 393.074,Z 919.45,A -85,B 0,C 180,E1 18285.943,E2 18285.943} C_VEL
LIN {X 0,Y 392.482,Z 926.841,A -85,B 0,C 180,E1 18282.803,E2 18282.803} C_VEL
LIN {X 0,Y 392.158,Z 932.197,A -85,B 0,C 180,E1 18279.834,E2 18279.834} C_VEL
LIN {X 0,Y 392.034,Z 936.026,A -85,B 0,C 180,E1 18277.03,E2 18277.03} C_VEL
LIN {X 0,Y 391.978,Z 938.836,A -85,B 0,C 180,E1 18273.801,E2 18273.801} C_VEL
LIN {X 0,Y 391.966,Z 939.894,A -85,B 0,C 180,E1 18271.022,E2 18271.022} C_VEL
LIN {X 0,Y 391.958,Z 939.763,A -85,B 0,C 180,E1 18268.244,E2 18268.244} C_VEL
LIN {X 0,Y 391.981,Z 938.015,A -85,B 0,C 180,E1 18265.023,E2 18265.023} C_VEL
LIN {X 0,Y 392.061,Z 935.158,A -85,B 0,C 180,E1 18262.23,E2 18262.23} C_VEL
LIN {X 0,Y 392.25,Z 930.329,A -85,B 0,C 180,E1 18258.977,E2 18258.977} C_VEL
LIN {X 0,Y 392.679,Z 924.204,A -85,B 0,C 180,E1 18255.959,E2 18255.959} C_VEL
LIN {X 0,Y 393.396,Z 916.474,A -85,B 0,C 180,E1 18252.852,E2 18252.852} C_VEL
LIN {X 0,Y 394.537,Z 906.678,A -85,B 0,C 180,E1 18249.683,E2 18249.683} C_VEL
LIN {X 0,Y 396.099,Z 895.691,A -85,B 0,C 180,E1 18246.651,E2 18246.651} C_VEL
LIN {X 0,Y 398.1,Z 883.318,A -85,B 0,C 180,E1 18243.765,E2 18243.765} C_VEL
LIN {X 0,Y 400.808,Z 868.191,A -85,B 0,C 180,E1 18240.728,E2 18240.728} C_VEL
LIN {X 0,Y 403.629,Z 853.324,A -85,B 0,C 180,E1 18238.153,E2 18238.153} C_VEL
LIN {X 0,Y 406.93,Z 836.475,A -85,B 0,C 180,E1 18235.647,E2 18235.647} C_VEL
LIN {X 0,Y 410.437,Z 818.736,A -85,B 0,C 180,E1 18233.355,E2 18233.355} C_VEL
LIN {X 0,Y 414.066,Z 799.869,A -85,B 0,C 180,E1 18231.286,E2 18231.286} C_VEL
LIN {X 0,Y 417.89,Z 778.885,A -85,B 0,C 180,E1 18229.329,E2 18229.329} C_VEL
LIN {X 0,Y 421.37,Z 758.527,A -85,B 0,C 180,E1 18227.731,E2 18227.731} C_VEL
LIN {X 0,Y 424.574,Z 737.313,A -85,B 0,C 180,E1 18226.368,E2 18226.368} C_VEL
LIN {X 0,Y 427.532,Z 715.193,A -85,B 0,C 180,E1 18225.207,E2 18225.207} C_VEL
LIN {X 0,Y 429.78,Z 694.513,A -85,B 0,C 180,E1 18224.354,E2 18224.354} C_VEL
LIN {X 0,Y 431.787,Z 670.814,A -85,B 0,C 180,E1 18223.625,E2 18223.625} C_VEL
LIN {X 0,Y 432.97,Z 647.857,A -85,B 0,C 180,E1 18223.131,E2 18223.131} C_VEL
LIN {X 0,Y 438.37,Z 449.14,A -85,B 0,C 180,E1 18219.632,E2 18219.632} C_VEL
LIN {X 0,Y 441.292,Z 347.111,A -85,B 0,C 180,E1 18217.763,E2 18217.763} C_VEL
LIN {X 0,Y 439.683,Z 330.206,A -85,B 0,C 180,E1 18217.181,E2 18217.181} C_VEL
LIN {X 0,Y 436.333,Z 324.902,A -85,B 0,C 180,E1 18216.569,E2 18216.569} C_VEL
LIN {X 0,Y 427.353,Z 307.579,A -85,B 0,C 180,E1 18213.838,E2 18213.838} C_VEL
LIN {X 0,Y 417.621,Z 290.082,A -85,B 0,C 180,E1 18210.661,E2 18210.661} C_VEL
LIN {X 0,Y 409.163,Z 275.766,A -85,B 0,C 180,E1 18207.665,E2 18207.665} C_VEL
LIN {X 0,Y 405.606,Z 270.169,A -85,B 0,C 180,E1 18206.342,E2 18206.342} C_VEL
LIN {X 0,Y 403.262,Z 266.061,A -85,B 0,C 180,E1 18205.401,E2 18205.401} C_VEL
LIN {X 0,Y 400.681,Z 262.086,A -85,B 0,C 180,E1 18204.379,E2 18204.379} C_VEL
LIN {X 0,Y 399.931,Z 260.723,A -85,B 0,C 180,E1 18204.049,E2 18204.049} C_VEL
LIN {X 0,Y 397.553,Z 257.4,A -85,B 0,C 180,E1 18203.101,E2 18203.101} C_VEL
LIN {X 0,Y 396.738,Z 255.498,A -85,B 0,C 180,E1 18202.681,E2 18202.681} C_VEL
LIN {X 0,Y 394.309,Z 252.609,A -85,B 0,C 180,E1 18201.729,E2 18201.729} C_VEL
LIN {X 0,Y 393.557,Z 250.356,A -85,B 0,C 180,E1 18201.147,E2 18201.147} C_VEL
LIN {X 0,Y 393.514,Z 250.014,A -85,B 0,C 180,E1 18199.442,E2 18199.442} C_VEL
LIN {X 0,Y 393.529,Z 250.014,A -85,B 0,C 180,E1 18195.624,E2 18195.624} C_VEL
LIN {X 0,Y 393.543,Z 250.017,A -85,B 0,C 180,E1 18191.728,E2 18191.728} C_VEL
LIN {X 0,Y 393.559,Z 250.023,A -85,B 0,C 180,E1 18187.739,E2 18187.739} C_VEL
LIN {X 0,Y 393.559,Z 250.023,A -85,B 0,C 180,E1 18183.788,E2 18183.788} C_VEL
LIN {X 0,Y 393.569,Z 250.008,A -85,B 0,C 180,E1 18179.709,E2 18179.709} C_VEL
LIN {X 0,Y 393.559,Z 249.998,A -85,B 0,C 180,E1 18175.629,E2 18175.629} C_VEL
LIN {X 0,Y 393.563,Z 249.995,A -85,B 0,C 180,E1 18171.674,E2 18171.674} C_VEL
LIN {X 0,Y 393.56,Z 250.015,A -85,B 0,C 180,E1 18167.679,E2 18167.679} C_VEL
LIN {X 0,Y 393.556,Z 250.023,A -85,B 0,C 180,E1 18163.773,E2 18163.773} C_VEL
LIN {X 0,Y 393.552,Z 250.001,A -85,B 0,C 180,E1 18159.787,E2 18159.787} C_VEL
LIN {X 0,Y 393.547,Z 249.998,A -85,B 0,C 180,E1 18155.856,E2 18155.856} C_VEL
LIN {X 0,Y 393.55,Z 250.011,A -85,B 0,C 180,E1 18151.837,E2 18151.837} C_VEL
LIN {X 0,Y 393.552,Z 250.026,A -85,B 0,C 180,E1 18147.929,E2 18147.929} C_VEL
LIN {X 0,Y 393.55,Z 250.014,A -85,B 0,C 180,E1 18143.885,E2 18143.885} C_VEL
LIN {X 0,Y 393.55,Z 249.999,A -85,B 0,C 180,E1 18139.884,E2 18139.884} C_VEL
LIN {X 0,Y 393.554,Z 249.999,A -85,B 0,C 180,E1 18135.885,E2 18135.885} C_VEL
LIN {X 0,Y 393.556,Z 250.002,A -85,B 0,C 180,E1 18131.895,E2 18131.895} C_VEL
LIN {X 0,Y 393.562,Z 250.005,A -85,B 0,C 180,E1 18127.939,E2 18127.939} C_VEL
LIN {X 0,Y 393.559,Z 250.006,A -85,B 0,C 180,E1 18123.983,E2 18123.983} C_VEL
LIN {X 0,Y 393.596,Z 250.259,A -85,B 0,C 180,E1 18121.556,E2 18121.556} C_VEL
LIN {X 0,Y 395.189,Z 253.956,A -85,B 0,C 180,E1 18120.568,E2 18120.568} C_VEL
LIN {X 0,Y 396.832,Z 255.942,A -85,B 0,C 180,E1 18119.92,E2 18119.92} C_VEL
LIN {X 0,Y 398.86,Z 259.73,A -85,B 0,C 180,E1 18118.973,E2 18118.973} C_VEL
LIN {X 0,Y 399.944,Z 261.365,A -85,B 0,C 180,E1 18118.524,E2 18118.524} C_VEL
LIN {X 0,Y 403.22,Z 267.211,A -85,B 0,C 180,E1 18117.103,E2 18117.103} C_VEL
LIN {X 0,Y 405.954,Z 272.008,A -85,B 0,C 180,E1 18115.977,E2 18115.977} C_VEL
LIN {X 0,Y 411.191,Z 281.458,A -85,B 0,C 180,E1 18113.898,E2 18113.898} C_VEL
LIN {X 0,Y 417.457,Z 293.505,A -85,B 0,C 180,E1 18111.498,E2 18111.498} C_VEL
LIN {X 0,Y 424.695,Z 308.587,A -85,B 0,C 180,E1 18108.818,E2 18108.818} C_VEL
LIN {X 0,Y 430.503,Z 322.165,A -85,B 0,C 180,E1 18106.67,E2 18106.67} C_VEL
LIN {X 0,Y 423.848,Z 377.584,A -85,B 0,C 180,E1 18102.467,E2 18102.467} C_VEL
LIN {X 0,Y 421.383,Z 400.843,A -85,B 0,C 180,E1 18100.748,E2 18100.748} C_VEL
LIN {X 0,Y 425.933,Z 447.216,A -85,B 0,C 180,E1 18099.091,E2 18099.091} C_VEL
LIN {X 0,Y 423.244,Z 518.042,A -85,B 0,C 180,E1 18097.751,E2 18097.751} C_VEL
LIN {X 0,Y 422.171,Z 525.725,A -85,B 0,C 180,E1 18097.692,E2 18097.692} C_VEL
LIN {X 0,Y 416.548,Z 546.19,A -85,B 0,C 180,E1 18097.847,E2 18097.847} C_VEL
LIN {X 0,Y 415.731,Z 552.78,A -85,B 0,C 180,E1 18097.783,E2 18097.783} C_VEL
LIN {X 0,Y 412.313,Z 634.945,A -85,B 0,C 180,E1 18096.131,E2 18096.131} C_VEL
LIN {X 0,Y 410.793,Z 655.122,A -85,B 0,C 180,E1 18095.48,E2 18095.48} C_VEL
LIN {X 0,Y 408.952,Z 673.842,A -85,B 0,C 180,E1 18094.629,E2 18094.629} C_VEL
LIN {X 0,Y 406.704,Z 692.374,A -85,B 0,C 180,E1 18093.525,E2 18093.525} C_VEL
LIN {X 0,Y 404.058,Z 710.811,A -85,B 0,C 180,E1 18092.129,E2 18092.129} C_VEL
LIN {X 0,Y 401.372,Z 727.43,A -85,B 0,C 180,E1 18090.572,E2 18090.572} C_VEL
LIN {X 0,Y 398.516,Z 743.694,A -85,B 0,C 180,E1 18088.708,E2 18088.708} C_VEL
LIN {X 0,Y 395.801,Z 758.317,A -85,B 0,C 180,E1 18086.671,E2 18086.671} C_VEL
LIN {X 0,Y 393.274,Z 771.462,A -85,B 0,C 180,E1 18084.458,E2 18084.458} C_VEL
LIN {X 0,Y 391.04,Z 783.168,A -85,B 0,C 180,E1 18082.065,E2 18082.065} C_VEL
LIN {X 0,Y 389.142,Z 793.439,A -85,B 0,C 180,E1 18079.491,E2 18079.491} C_VEL
LIN {X 0,Y 387.694,Z 801.81,A -85,B 0,C 180,E1 18076.884,E2 18076.884} C_VEL
LIN {X 0,Y 386.619,Z 808.794,A -85,B 0,C 180,E1 18074.091,E2 18074.091} C_VEL
LIN {X 0,Y 385.91,Z 814.035,A -85,B 0,C 180,E1 18071.262,E2 18071.262} C_VEL
LIN {X 0,Y 385.52,Z 817.599,A -85,B 0,C 180,E1 18068.392,E2 18068.392} C_VEL
LIN {X 0,Y 385.363,Z 819.516,A -85,B 0,C 180,E1 18065.474,E2 18065.474} C_VEL
LIN {X 0,Y 385.391,Z 819.754,A -85,B 0,C 180,E1 18062.499,E2 18062.499} C_VEL
LIN {X 0,Y 385.609,Z 818.33,A -85,B 0,C 180,E1 18059.63,E2 18059.63} C_VEL
LIN {X 0,Y 386.082,Z 815.179,A -85,B 0,C 180,E1 18056.702,E2 18056.702} C_VEL
LIN {X 0,Y 386.937,Z 810.121,A -85,B 0,C 180,E1 18053.722,E2 18053.722} C_VEL
LIN {X 0,Y 388.187,Z 803.266,A -85,B 0,C 180,E1 18050.83,E2 18050.83} C_VEL
LIN {X 0,Y 389.928,Z 794.594,A -85,B 0,C 180,E1 18048.039,E2 18048.039} C_VEL
LIN {X 0,Y 392.039,Z 784.55,A -85,B 0,C 180,E1 18045.466,E2 18045.466} C_VEL
LIN {X 0,Y 394.46,Z 773.303,A -85,B 0,C 180,E1 18043.116,E2 18043.116} C_VEL
LIN {X 0,Y 397.257,Z 760.262,A -85,B 0,C 180,E1 18040.873,E2 18040.873} C_VEL
LIN {X 0,Y 400.263,Z 745.647,A -85,B 0,C 180,E1 18038.8,E2 18038.8} C_VEL
LIN {X 0,Y 403.361,Z 729.589,A -85,B 0,C 180,E1 18036.929,E2 18036.929} C_VEL
LIN {X 0,Y 406.389,Z 712.678,A -85,B 0,C 180,E1 18035.322,E2 18035.322} C_VEL
LIN {X 0,Y 409.283,Z 694.237,A -85,B 0,C 180,E1 18033.906,E2 18033.906} C_VEL
LIN {X 0,Y 411.794,Z 675.696,A -85,B 0,C 180,E1 18032.782,E2 18032.782} C_VEL
LIN {X 0,Y 413.973,Z 655.735,A -85,B 0,C 180,E1 18031.863,E2 18031.863} C_VEL
LIN {X 0,Y 415.662,Z 635.387,A -85,B 0,C 180,E1 18031.204,E2 18031.204} C_VEL
LIN {X 0,Y 422.603,Z 496.402,A -85,B 0,C 180,E1 18028.341,E2 18028.341} C_VEL
LIN {X 0,Y 424.841,Z 447.938,A -85,B 0,C 180,E1 18027.36,E2 18027.36} C_VEL
LIN {X 0,Y 420.054,Z 394.319,A -85,B 0,C 180,E1 18025.18,E2 18025.18} C_VEL
LIN {X 0,Y 420.312,Z 390.054,A -85,B 0,C 180,E1 18024.9,E2 18024.9} C_VEL
LIN {X 0,Y 427.744,Z 337.564,A -85,B 0,C 180,E1 18020.811,E2 18020.811} C_VEL
LIN {X 0,Y 428.754,Z 330.64,A -85,B 0,C 180,E1 18020.261,E2 18020.261} C_VEL
LIN {X 0,Y 421.981,Z 315.023,A -85,B 0,C 180,E1 18017.37,E2 18017.37} C_VEL
LIN {X 0,Y 415.625,Z 301.685,A -85,B 0,C 180,E1 18014.488,E2 18014.488} C_VEL
LIN {X 0,Y 410.649,Z 292.277,A -85,B 0,C 180,E1 18012.086,E2 18012.086} C_VEL
LIN {X 0,Y 408.029,Z 287.547,A -85,B 0,C 180,E1 18010.733,E2 18010.733} C_VEL
LIN {X 0,Y 405.836,Z 283.494,A -85,B 0,C 180,E1 18009.501,E2 18009.501} C_VEL
LIN {X 0,Y 403.018,Z 278.605,A -85,B 0,C 180,E1 18007.842,E2 18007.842} C_VEL
LIN {X 0,Y 400.703,Z 274.429,A -85,B 0,C 180,E1 18006.303,E2 18006.303} C_VEL
LIN {X 0,Y 397.827,Z 270.113,A -85,B 0,C 180,E1 18004.324,E2 18004.324} C_VEL
LIN {X 0,Y 397.243,Z 268.668,A -85,B 0,C 180,E1 18003.752,E2 18003.752} C_VEL
LIN {X 0,Y 394.494,Z 265.186,A -85,B 0,C 180,E1 18001.597,E2 18001.597} C_VEL
LIN {X 0,Y 393.619,Z 262.963,A -85,B 0,C 180,E1 18000.436,E2 18000.436} C_VEL
LIN {X 0,Y 390.467,Z 259.016,A -85,B 0,C 180,E1 17996.476,E2 17996.476} C_VEL
LIN {X 0,Y 389.692,Z 257.161,A -85,B 0,C 180,E1 17994.109,E2 17994.109} C_VEL
LIN {X 0,Y 389.299,Z 256.838,A -85,B 0,C 180,E1 17990.091,E2 17990.091} C_VEL
LIN {X 0,Y 390.111,Z 257.818,A -85,B 0,C 180,E1 17987.416,E2 17987.416} C_VEL
LIN {X 0,Y 393.091,Z 262.577,A -85,B 0,C 180,E1 17982.839,E2 17982.839} C_VEL
LIN {X 0,Y 394.243,Z 263.746,A -85,B 0,C 180,E1 17981.823,E2 17981.823} C_VEL
LIN {X 0,Y 396.373,Z 267.735,A -85,B 0,C 180,E1 17979.782,E2 17979.782} C_VEL
LIN {X 0,Y 397.976,Z 269.294,A -85,B 0,C 180,E1 17978.756,E2 17978.756} C_VEL
LIN {X 0,Y 399.823,Z 273.021,A -85,B 0,C 180,E1 17977.33,E2 17977.33} C_VEL
LIN {X 0,Y 401.512,Z 275.105,A -85,B 0,C 180,E1 17976.363,E2 17976.363} C_VEL
LIN {X 0,Y 403.889,Z 279.107,A -85,B 0,C 180,E1 17974.955,E2 17974.955} C_VEL
LIN {X 0,Y 405.2,Z 281.31,A -85,B 0,C 180,E1 17974.24,E2 17974.24} C_VEL
LIN {X 0,Y 407.994,Z 285.881,A -85,B 0,C 180,E1 17972.818,E2 17972.818} C_VEL
LIN {X 0,Y 411.055,Z 291.133,A -85,B 0,C 180,E1 17971.367,E2 17971.367} C_VEL
LIN {X 0,Y 415.719,Z 299.356,A -85,B 0,C 180,E1 17969.343,E2 17969.343} C_VEL
LIN {X 0,Y 422.097,Z 311.429,A -85,B 0,C 180,E1 17966.825,E2 17966.825} C_VEL
LIN {X 0,Y 428.9,Z 325.49,A -85,B 0,C 180,E1 17964.352,E2 17964.352} C_VEL
LIN {X 0,Y 432.111,Z 332.287,A -85,B 0,C 180,E1 17963.346,E2 17963.346} C_VEL
LIN {X 0,Y 432.796,Z 333.908,A -85,B 0,C 180,E1 17963.212,E2 17963.212} C_VEL
LIN {X 0,Y 433.962,Z 351.231,A -85,B 0,C 180,E1 17962.653,E2 17962.653} C_VEL
LIN {X 0,Y 428.268,Z 546.485,A -85,B 0,C 180,E1 17959.135,E2 17959.135} C_VEL
LIN {X 0,Y 425.27,Z 659.799,A -85,B 0,C 180,E1 17957.148,E2 17957.148} C_VEL
LIN {X 0,Y 423.582,Z 682.545,A -85,B 0,C 180,E1 17956.549,E2 17956.549} C_VEL
LIN {X 0,Y 421.345,Z 705.079,A -85,B 0,C 180,E1 17955.727,E2 17955.727} C_VEL
LIN {X 0,Y 418.656,Z 726.587,A -85,B 0,C 180,E1 17954.699,E2 17954.699} C_VEL
LIN {X 0,Y 415.528,Z 747.921,A -85,B 0,C 180,E1 17953.422,E2 17953.422} C_VEL
LIN {X 0,Y 412.109,Z 768.825,A -85,B 0,C 180,E1 17951.911,E2 17951.911} C_VEL
LIN {X 0,Y 408.463,Z 788.688,A -85,B 0,C 180,E1 17950.173,E2 17950.173} C_VEL
LIN {X 0,Y 404.562,Z 808.91,A -85,B 0,C 180,E1 17948.094,E2 17948.094} C_VEL
LIN {X 0,Y 401.047,Z 826.665,A -85,B 0,C 180,E1 17945.951,E2 17945.951} C_VEL
LIN {X 0,Y 397.434,Z 844.546,A -85,B 0,C 180,E1 17943.43,E2 17943.43} C_VEL
LIN {X 0,Y 394.293,Z 860.648,A -85,B 0,C 180,E1 17940.811,E2 17940.811} C_VEL
LIN {X 0,Y 391.521,Z 875.281,A -85,B 0,C 180,E1 17938.025,E2 17938.025} C_VEL
LIN {X 0,Y 389.038,Z 889.53,A -85,B 0,C 180,E1 17934.873,E2 17934.873} C_VEL
LIN {X 0,Y 387.315,Z 900.719,A -85,B 0,C 180,E1 17931.98,E2 17931.98} C_VEL
LIN {X 0,Y 385.911,Z 911.298,A -85,B 0,C 180,E1 17928.738,E2 17928.738} C_VEL
LIN {X 0,Y 385.058,Z 919.282,A -85,B 0,C 180,E1 17925.82,E2 17925.82} C_VEL
LIN {X 0,Y 384.483,Z 926.686,A -85,B 0,C 180,E1 17922.463,E2 17922.463} C_VEL
LIN {X 0,Y 384.197,Z 931.775,A -85,B 0,C 180,E1 17919.483,E2 17919.483} C_VEL
LIN {X 0,Y 384.099,Z 935.732,A -85,B 0,C 180,E1 17916.275,E2 17916.275} C_VEL
LIN {X 0,Y 384.064,Z 937.916,A -85,B 0,C 180,E1 17913.282,E2 17913.282} C_VEL
LIN {X 0,Y 384.051,Z 938.799,A -85,B 0,C 180,E1 17910.297,E2 17910.297} C_VEL
LIN {X 0,Y 384.061,Z 938.09,A -85,B 0,C 180,E1 17907.014,E2 17907.014} C_VEL
LIN {X 0,Y 384.073,Z 936.158,A -85,B 0,C 180,E1 17904.171,E2 17904.171} C_VEL
LIN {X 0,Y 384.149,Z 932.623,A -85,B 0,C 180,E1 17901.014,E2 17901.014} C_VEL
LIN {X 0,Y 384.416,Z 927.598,A -85,B 0,C 180,E1 17897.951,E2 17897.951} C_VEL
LIN {X 0,Y 384.878,Z 921.354,A -85,B 0,C 180,E1 17894.941,E2 17894.941} C_VEL
LIN {X 0,Y 385.757,Z 912.95,A -85,B 0,C 180,E1 17891.721,E2 17891.721} C_VEL
LIN {X 0,Y 387.008,Z 903.356,A -85,B 0,C 180,E1 17888.635,E2 17888.635} C_VEL
LIN {X 0,Y 388.783,Z 891.829,A -85,B 0,C 180,E1 17885.539,E2 17885.539} C_VEL
LIN {X 0,Y 391.102,Z 878.774,A -85,B 0,C 180,E1 17882.513,E2 17882.513} C_VEL
LIN {X 0,Y 393.852,Z 864.228,A -85,B 0,C 180,E1 17879.654,E2 17879.654} C_VEL
LIN {X 0,Y 397.265,Z 847.416,A -85,B 0,C 180,E1 17876.809,E2 17876.809} C_VEL
LIN {X 0,Y 400.744,Z 830.68,A -85,B 0,C 180,E1 17874.366,E2 17874.366} C_VEL
LIN {X 0,Y 404.368,Z 813.081,A -85,B 0,C 180,E1 17872.176,E2 17872.176} C_VEL
LIN {X 0,Y 408.073,Z 794.627,A -85,B 0,C 180,E1 17870.186,E2 17870.186} C_VEL
LIN {X 0,Y 411.728,Z 775.112,A -85,B 0,C 180,E1 17868.414,E2 17868.414} C_VEL
LIN {X 0,Y 415.441,Z 753.959,A -85,B 0,C 180,E1 17866.795,E2 17866.795} C_VEL
LIN {X 0,Y 418.473,Z 734.611,A -85,B 0,C 180,E1 17865.566,E2 17865.566} C_VEL
LIN {X 0,Y 421.482,Z 712.186,A -85,B 0,C 180,E1 17864.412,E2 17864.412} C_VEL
LIN {X 0,Y 423.898,Z 690.449,A -85,B 0,C 180,E1 17863.534,E2 17863.534} C_VEL
LIN {X 0,Y 425.759,Z 667.76,A -85,B 0,C 180,E1 17862.873,E2 17862.873} C_VEL
LIN {X 0,Y 426.956,Z 641.751,A -85,B 0,C 180,E1 17862.344,E2 17862.344} C_VEL
LIN {X 0,Y 432.583,Z 446.366,A -85,B 0,C 180,E1 17858.862,E2 17858.862} C_VEL
LIN {X 0,Y 435.548,Z 348.457,A -85,B 0,C 180,E1 17857.052,E2 17857.052} C_VEL
LIN {X 0,Y 434.208,Z 334.319,A -85,B 0,C 180,E1 17856.551,E2 17856.551} C_VEL
LIN {X 0,Y 429.049,Z 326.375,A -85,B 0,C 180,E1 17855.634,E2 17855.634} C_VEL
LIN {X 0,Y 420.236,Z 309.471,A -85,B 0,C 180,E1 17852.853,E2 17852.853} C_VEL
LIN {X 0,Y 410.73,Z 292.385,A -85,B 0,C 180,E1 17849.615,E2 17849.615} C_VEL
LIN {X 0,Y 402.126,Z 277.816,A -85,B 0,C 180,E1 17846.428,E2 17846.428} C_VEL
LIN {X 0,Y 399.213,Z 273.101,A -85,B 0,C 180,E1 17845.289,E2 17845.289} C_VEL
LIN {X 0,Y 396.033,Z 267.989,A -85,B 0,C 180,E1 17843.984,E2 17843.984} C_VEL
LIN {X 0,Y 393.026,Z 263.533,A -85,B 0,C 180,E1 17842.749,E2 17842.749} C_VEL
LIN {X 0,Y 392.156,Z 261.837,A -85,B 0,C 180,E1 17842.328,E2 17842.328} C_VEL
LIN {X 0,Y 389.592,Z 258.169,A -85,B 0,C 180,E1 17841.215,E2 17841.215} C_VEL
LIN {X 0,Y 388.789,Z 256.491,A -85,B 0,C 180,E1 17840.788,E2 17840.788} C_VEL
LIN {X 0,Y 386.46,Z 253.754,A -85,B 0,C 180,E1 17839.812,E2 17839.812} C_VEL
LIN {X 0,Y 385.618,Z 251.318,A -85,B 0,C 180,E1 17839.148,E2 17839.148} C_VEL
LIN {X 0,Y 385.574,Z 251.01,A -85,B 0,C 180,E1 17837.04,E2 17837.04} C_VEL
LIN {X 0,Y 385.575,Z 251.009,A -85,B 0,C 180,E1 17833.039,E2 17833.039} C_VEL
LIN {X 0,Y 385.578,Z 251.005,A -85,B 0,C 180,E1 17828.951,E2 17828.951} C_VEL
LIN {X 0,Y 385.582,Z 250.996,A -85,B 0,C 180,E1 17824.909,E2 17824.909} C_VEL
LIN {X 0,Y 385.584,Z 250.988,A -85,B 0,C 180,E1 17820.892,E2 17820.892} C_VEL
LIN {X 0,Y 385.59,Z 250.991,A -85,B 0,C 180,E1 17816.863,E2 17816.863} C_VEL
LIN {X 0,Y 385.596,Z 251.006,A -85,B 0,C 180,E1 17812.851,E2 17812.851} C_VEL
LIN {X 0,Y 385.601,Z 251.015,A -85,B 0,C 180,E1 17808.787,E2 17808.787} C_VEL
LIN {X 0,Y 385.607,Z 250.994,A -85,B 0,C 180,E1 17804.819,E2 17804.819} C_VEL
LIN {X 0,Y 385.618,Z 250.982,A -85,B 0,C 180,E1 17800.932,E2 17800.932} C_VEL
LIN {X 0,Y 385.626,Z 250.998,A -85,B 0,C 180,E1 17796.952,E2 17796.952} C_VEL
LIN {X 0,Y 385.627,Z 251.013,A -85,B 0,C 180,E1 17792.792,E2 17792.792} C_VEL
LIN {X 0,Y 385.624,Z 251.001,A -85,B 0,C 180,E1 17788.765,E2 17788.765} C_VEL
LIN {X 0,Y 385.618,Z 250.988,A -85,B 0,C 180,E1 17784.676,E2 17784.676} C_VEL
LIN {X 0,Y 385.617,Z 250.985,A -85,B 0,C 180,E1 17780.754,E2 17780.754} C_VEL
LIN {X 0,Y 385.618,Z 250.993,A -85,B 0,C 180,E1 17776.77,E2 17776.77} C_VEL
LIN {X 0,Y 385.617,Z 251.003,A -85,B 0,C 180,E1 17772.793,E2 17772.793} C_VEL
LIN {X 0,Y 385.615,Z 251.006,A -85,B 0,C 180,E1 17768.699,E2 17768.699} C_VEL
LIN {X 0,Y 385.613,Z 251.004,A -85,B 0,C 180,E1 17764.602,E2 17764.602} C_VEL
LIN {X 0,Y 385.67,Z 251.325,A -85,B 0,C 180,E1 17763.408,E2 17763.408} C_VEL
LIN {X 0,Y 387.235,Z 254.921,A -85,B 0,C 180,E1 17762.402,E2 17762.402} C_VEL
LIN {X 0,Y 388.949,Z 256.89,A -85,B 0,C 180,E1 17761.693,E2 17761.693} C_VEL
LIN {X 0,Y 390.812,Z 260.565,A -85,B 0,C 180,E1 17760.727,E2 17760.727} C_VEL
LIN {X 0,Y 392.185,Z 262.421,A -85,B 0,C 180,E1 17760.15,E2 17760.15} C_VEL
LIN {X 0,Y 394.609,Z 266.519,A -85,B 0,C 180,E1 17759.056,E2 17759.056} C_VEL
LIN {X 0,Y 400.789,Z 277.494,A -85,B 0,C 180,E1 17756.365,E2 17756.365} C_VEL
LIN {X 0,Y 407.819,Z 290.399,A -85,B 0,C 180,E1 17753.519,E2 17753.519} C_VEL
LIN {X 0,Y 415.937,Z 306.825,A -85,B 0,C 180,E1 17750.366,E2 17750.366} C_VEL
LIN {X 0,Y 423.702,Z 324.228,A -85,B 0,C 180,E1 17747.441,E2 17747.441} C_VEL
LIN {X 0,Y 424.3,Z 325.811,A -85,B 0,C 180,E1 17747.203,E2 17747.203} C_VEL
LIN {X 0,Y 417.32,Z 381.29,A -85,B 0,C 180,E1 17742.946,E2 17742.946} C_VEL
LIN {X 0,Y 415.277,Z 400.02,A -85,B 0,C 180,E1 17741.556,E2 17741.556} C_VEL
LIN {X 0,Y 419.894,Z 448.296,A -85,B 0,C 180,E1 17739.791,E2 17739.791} C_VEL
LIN {X 0,Y 415.731,Z 552.78,A -85,B 0,C 180,E1 17737.783,E2 17737.783} C_VEL
LIN {X 0,Y 414.681,Z 560.457,A -85,B 0,C 180,E1 17737.719,E2 17737.719} C_VEL
LIN {X 0,Y 409,Z 580.908,A -85,B 0,C 180,E1 17737.876,E2 17737.876} C_VEL
LIN {X 0,Y 408.136,Z 587.497,A -85,B 0,C 180,E1 17737.812,E2 17737.812} C_VEL
LIN {X 0,Y 405.94,Z 636.043,A -85,B 0,C 180,E1 17736.796,E2 17736.796} C_VEL
LIN {X 0,Y 404.355,Z 656.016,A -85,B 0,C 180,E1 17736.136,E2 17736.136} C_VEL
LIN {X 0,Y 402.334,Z 675.447,A -85,B 0,C 180,E1 17735.23,E2 17735.23} C_VEL
LIN {X 0,Y 399.958,Z 693.982,A -85,B 0,C 180,E1 17734.096,E2 17734.096} C_VEL
LIN {X 0,Y 397.316,Z 711.561,A -85,B 0,C 180,E1 17732.742,E2 17732.742} C_VEL
LIN {X 0,Y 394.501,Z 728.196,A -85,B 0,C 180,E1 17731.163,E2 17731.163} C_VEL
LIN {X 0,Y 391.496,Z 744.488,A -85,B 0,C 180,E1 17729.27,E2 17729.27} C_VEL
LIN {X 0,Y 388.633,Z 759.145,A -85,B 0,C 180,E1 17727.2,E2 17727.2} C_VEL
LIN {X 0,Y 385.96,Z 772.328,A -85,B 0,C 180,E1 17724.948,E2 17724.948} C_VEL
LIN {X 0,Y 383.583,Z 784.078,A -85,B 0,C 180,E1 17722.513,E2 17722.513} C_VEL
LIN {X 0,Y 381.559,Z 794.392,A -85,B 0,C 180,E1 17719.89,E2 17719.89} C_VEL
LIN {X 0,Y 380.004,Z 802.806,A -85,B 0,C 180,E1 17717.233,E2 17717.233} C_VEL
LIN {X 0,Y 378.842,Z 809.837,A -85,B 0,C 180,E1 17714.385,E2 17714.385} C_VEL
LIN {X 0,Y 378.073,Z 815.121,A -85,B 0,C 180,E1 17711.499,E2 17711.499} C_VEL
LIN {X 0,Y 377.634,Z 818.733,A -85,B 0,C 180,E1 17708.571,E2 17708.571} C_VEL
LIN {X 0,Y 377.46,Z 820.701,A -85,B 0,C 180,E1 17705.594,E2 17705.594} C_VEL
LIN {X 0,Y 377.485,Z 821.002,A -85,B 0,C 180,E1 17702.537,E2 17702.537} C_VEL
LIN {X 0,Y 377.714,Z 819.644,A -85,B 0,C 180,E1 17699.631,E2 17699.631} C_VEL
LIN {X 0,Y 378.213,Z 816.577,A -85,B 0,C 180,E1 17696.644,E2 17696.644} C_VEL
LIN {X 0,Y 379.049,Z 811.948,A -85,B 0,C 180,E1 17693.784,E2 17693.784} C_VEL
LIN {X 0,Y 380.218,Z 805.899,A -85,B 0,C 180,E1 17691.063,E2 17691.063} C_VEL
LIN {X 0,Y 381.893,Z 797.992,A -85,B 0,C 180,E1 17688.319,E2 17688.319} C_VEL
LIN {X 0,Y 383.985,Z 788.623,A -85,B 0,C 180,E1 17685.73,E2 17685.73} C_VEL
LIN {X 0,Y 386.586,Z 777.199,A -85,B 0,C 180,E1 17683.17,E2 17683.17} C_VEL
LIN {X 0,Y 389.403,Z 764.823,A -85,B 0,C 180,E1 17680.9,E2 17680.9} C_VEL
LIN {X 0,Y 392.615,Z 750.214,A -85,B 0,C 180,E1 17678.692,E2 17678.692} C_VEL
LIN {X 0,Y 395.831,Z 734.77,A -85,B 0,C 180,E1 17676.773,E2 17676.773} C_VEL
LIN {X 0,Y 398.988,Z 718.359,A -85,B 0,C 180,E1 17675.098,E2 17675.098} C_VEL
LIN {X 0,Y 402.108,Z 700.197,A -85,B 0,C 180,E1 17673.596,E2 17673.596} C_VEL
LIN {X 0,Y 404.869,Z 681.584,A -85,B 0,C 180,E1 17672.375,E2 17672.375} C_VEL
LIN {X 0,Y 407.296,Z 661.621,A -85,B 0,C 180,E1 17671.368,E2 17671.368} C_VEL
LIN {X 0,Y 409.226,Z 641.23,A -85,B 0,C 180,E1 17670.627,E2 17670.627} C_VEL
LIN {X 0,Y 410.849,Z 614.903,A -85,B 0,C 180,E1 17670.003,E2 17670.003} C_VEL
LIN {X 0,Y 419.303,Z 449.777,A -85,B 0,C 180,E1 17666.617,E2 17666.617} C_VEL
LIN {X 0,Y 414.743,Z 395.72,A -85,B 0,C 180,E1 17664.374,E2 17664.374} C_VEL
LIN {X 0,Y 414.5,Z 390.907,A -85,B 0,C 180,E1 17664.133,E2 17664.133} C_VEL
LIN {X 0,Y 422.248,Z 338.845,A -85,B 0,C 180,E1 17660.034,E2 17660.034} C_VEL
LIN {X 0,Y 422.812,Z 334.747,A -85,B 0,C 180,E1 17659.692,E2 17659.692} C_VEL
LIN {X 0,Y 416.541,Z 319.93,A -85,B 0,C 180,E1 17656.884,E2 17656.884} C_VEL
LIN {X 0,Y 410.621,Z 307.368,A -85,B 0,C 180,E1 17654.092,E2 17654.092} C_VEL
LIN {X 0,Y 406.067,Z 298.502,A -85,B 0,C 180,E1 17651.792,E2 17651.792} C_VEL
LIN {X 0,Y 401.907,Z 290.513,A -85,B 0,C 180,E1 17649.45,E2 17649.45} C_VEL
LIN {X 0,Y 398.879,Z 285.306,A -85,B 0,C 180,E1 17647.634,E2 17647.634} C_VEL
LIN {X 0,Y 396.175,Z 280.554,A -85,B 0,C 180,E1 17645.793,E2 17645.793} C_VEL
LIN {X 0,Y 393.875,Z 276.859,A -85,B 0,C 180,E1 17644.075,E2 17644.075} C_VEL
LIN {X 0,Y 393.258,Z 275.517,A -85,B 0,C 180,E1 17643.498,E2 17643.498} C_VEL
LIN {X 0,Y 390.697,Z 271.975,A -85,B 0,C 180,E1 17641.319,E2 17641.319} C_VEL
LIN {X 0,Y 389.934,Z 270.033,A -85,B 0,C 180,E1 17640.28,E2 17640.28} C_VEL
LIN {X 0,Y 386.998,Z 266.271,A -85,B 0,C 180,E1 17636.444,E2 17636.444} C_VEL
LIN {X 0,Y 386.321,Z 264.438,A -85,B 0,C 180,E1 17634.206,E2 17634.206} C_VEL
LIN {X 0,Y 385.93,Z 264.09,A -85,B 0,C 180,E1 17630.154,E2 17630.154} C_VEL
LIN {X 0,Y 386.717,Z 265.069,A -85,B 0,C 180,E1 17627.456,E2 17627.456} C_VEL
LIN {X 0,Y 389.718,Z 269.838,A -85,B 0,C 180,E1 17622.839,E2 17622.839} C_VEL
LIN {X 0,Y 390.653,Z 270.934,A -85,B 0,C 180,E1 17621.959,E2 17621.959} C_VEL
LIN {X 0,Y 392.986,Z 275.063,A -85,B 0,C 180,E1 17619.756,E2 17619.756} C_VEL
LIN {X 0,Y 394.268,Z 276.494,A -85,B 0,C 180,E1 17618.893,E2 17618.893} C_VEL
LIN {X 0,Y 396.415,Z 280.393,A -85,B 0,C 180,E1 17617.3,E2 17617.3} C_VEL
LIN {X 0,Y 397.602,Z 281.961,A -85,B 0,C 180,E1 17616.589,E2 17616.589} C_VEL
LIN {X 0,Y 400.24,Z 286.236,A -85,B 0,C 180,E1 17615.027,E2 17615.027} C_VEL
LIN {X 0,Y 404.106,Z 293.058,A -85,B 0,C 180,E1 17612.918,E2 17612.918} C_VEL
LIN {X 0,Y 408.516,Z 300.509,A -85,B 0,C 180,E1 17610.852,E2 17610.852} C_VEL
LIN {X 0,Y 415.34,Z 313.495,A -85,B 0,C 180,E1 17607.924,E2 17607.924} C_VEL
LIN {X 0,Y 422.041,Z 327.275,A -85,B 0,C 180,E1 17605.348,E2 17605.348} C_VEL
LIN {X 0,Y 425.077,Z 333.621,A -85,B 0,C 180,E1 17604.335,E2 17604.335} C_VEL
LIN {X 0,Y 427.481,Z 337.811,A -85,B 0,C 180,E1 17603.879,E2 17603.879} C_VEL
LIN {X 0,Y 428.389,Z 352.574,A -85,B 0,C 180,E1 17603.401,E2 17603.401} C_VEL
LIN {X 0,Y 422.433,Z 544.114,A -85,B 0,C 180,E1 17599.908,E2 17599.908} C_VEL
LIN {X 0,Y 419.179,Z 659.749,A -85,B 0,C 180,E1 17597.855,E2 17597.855} C_VEL
LIN {X 0,Y 417.428,Z 682.386,A -85,B 0,C 180,E1 17597.252,E2 17597.252} C_VEL
LIN {X 0,Y 415.081,Z 704.922,A -85,B 0,C 180,E1 17596.421,E2 17596.421} C_VEL
LIN {X 0,Y 412.36,Z 725.748,A -85,B 0,C 180,E1 17595.417,E2 17595.417} C_VEL
LIN {X 0,Y 409.118,Z 746.855,A -85,B 0,C 180,E1 17594.146,E2 17594.146} C_VEL
LIN {X 0,Y 405.665,Z 767.13,A -85,B 0,C 180,E1 17592.67,E2 17592.67} C_VEL
LIN {X 0,Y 401.998,Z 786.35,A -85,B 0,C 180,E1 17590.988,E2 17590.988} C_VEL
LIN {X 0,Y 398.077,Z 805.84,A -85,B 0,C 180,E1 17588.994,E2 17588.994} C_VEL
LIN {X 0,Y 394.236,Z 824.238,A -85,B 0,C 180,E1 17586.763,E2 17586.763} C_VEL
LIN {X 0,Y 390.35,Z 842.545,A -85,B 0,C 180,E1 17584.173,E2 17584.173} C_VEL
LIN {X 0,Y 386.953,Z 859.032,A -85,B 0,C 180,E1 17581.461,E2 17581.461} C_VEL
LIN {X 0,Y 384.004,Z 873.717,A -85,B 0,C 180,E1 17578.624,E2 17578.624} C_VEL
LIN {X 0,Y 381.416,Z 887.836,A -85,B 0,C 180,E1 17575.46,E2 17575.46} C_VEL
LIN {X 0,Y 379.543,Z 899.271,A -85,B 0,C 180,E1 17572.455,E2 17572.455} C_VEL
LIN {X 0,Y 378.048,Z 909.911,A -85,B 0,C 180,E1 17569.143,E2 17569.143} C_VEL
LIN {X 0,Y 377.158,Z 917.931,A -85,B 0,C 180,E1 17566.16,E2 17566.16} C_VEL
LIN {X 0,Y 376.552,Z 925.382,A -85,B 0,C 180,E1 17562.73,E2 17562.73} C_VEL
LIN {X 0,Y 376.269,Z 930.341,A -85,B 0,C 180,E1 17559.79,E2 17559.79} C_VEL
LIN {X 0,Y 376.181,Z 934.488,A -85,B 0,C 180,E1 17556.408,E2 17556.408} C_VEL
LIN {X 0,Y 376.152,Z 936.687,A -85,B 0,C 180,E1 17553.351,E2 17553.351} C_VEL
LIN {X 0,Y 376.141,Z 937.558,A -85,B 0,C 180,E1 17550.455,E2 17550.455} C_VEL
LIN {X 0,Y 376.148,Z 936.951,A -85,B 0,C 180,E1 17547.104,E2 17547.104} C_VEL
LIN {X 0,Y 376.149,Z 935.068,A -85,B 0,C 180,E1 17544.201,E2 17544.201} C_VEL
LIN {X 0,Y 376.207,Z 931.617,A -85,B 0,C 180,E1 17540.977,E2 17540.977} C_VEL
LIN {X 0,Y 376.481,Z 926.422,A -85,B 0,C 180,E1 17537.732,E2 17537.732} C_VEL
LIN {X 0,Y 376.959,Z 920.093,A -85,B 0,C 180,E1 17534.617,E2 17534.617} C_VEL
LIN {X 0,Y 377.882,Z 911.604,A -85,B 0,C 180,E1 17531.307,E2 17531.307} C_VEL
LIN {X 0,Y 379.23,Z 901.918,A -85,B 0,C 180,E1 17528.135,E2 17528.135} C_VEL
LIN {X 0,Y 381.097,Z 890.469,A -85,B 0,C 180,E1 17525.012,E2 17525.012} C_VEL
LIN {X 0,Y 383.493,Z 877.737,A -85,B 0,C 180,E1 17522.01,E2 17522.01} C_VEL
LIN {X 0,Y 386.322,Z 863.581,A -85,B 0,C 180,E1 17519.171,E2 17519.171} C_VEL
LIN {X 0,Y 389.885,Z 846.901,A -85,B 0,C 180,E1 17516.283,E2 17516.283} C_VEL
LIN {X 0,Y 393.306,Z 831.176,A -85,B 0,C 180,E1 17513.942,E2 17513.942} C_VEL
LIN {X 0,Y 397.33,Z 812.544,A -85,B 0,C 180,E1 17511.568,E2 17511.568} C_VEL
LIN {X 0,Y 401.266,Z 793.876,A -85,B 0,C 180,E1 17509.525,E2 17509.525} C_VEL
LIN {X 0,Y 405.083,Z 774.457,A -85,B 0,C 180,E1 17507.74,E2 17507.74} C_VEL
LIN {X 0,Y 408.905,Z 753.561,A -85,B 0,C 180,E1 17506.123,E2 17506.123} C_VEL
LIN {X 0,Y 411.889,Z 735.194,A -85,B 0,C 180,E1 17504.943,E2 17504.943} C_VEL
LIN {X 0,Y 415.04,Z 712.882,A -85,B 0,C 180,E1 17503.769,E2 17503.769} C_VEL
LIN {X 0,Y 417.472,Z 692.008,A -85,B 0,C 180,E1 17502.908,E2 17502.908} C_VEL
LIN {X 0,Y 419.509,Z 668.959,A -85,B 0,C 180,E1 17502.209,E2 17502.209} C_VEL
LIN {X 0,Y 420.741,Z 645.527,A -85,B 0,C 180,E1 17501.709,E2 17501.709} C_VEL
LIN {X 0,Y 426.743,Z 446.489,A -85,B 0,C 180,E1 17498.131,E2 17498.131} C_VEL
LIN {X 0,Y 429.852,Z 349.669,A -85,B 0,C 180,E1 17496.319,E2 17496.319} C_VEL
LIN {X 0,Y 428.84,Z 338.516,A -85,B 0,C 180,E1 17495.922,E2 17495.922} C_VEL
LIN {X 0,Y 421.374,Z 327.116,A -85,B 0,C 180,E1 17494.549,E2 17494.549} C_VEL
LIN {X 0,Y 412.404,Z 310.038,A -85,B 0,C 180,E1 17491.58,E2 17491.58} C_VEL
LIN {X 0,Y 403.108,Z 293.552,A -85,B 0,C 180,E1 17488.278,E2 17488.278} C_VEL
LIN {X 0,Y 396.378,Z 282.506,A -85,B 0,C 180,E1 17485.714,E2 17485.714} C_VEL
LIN {X 0,Y 393.634,Z 277.953,A -85,B 0,C 180,E1 17484.583,E2 17484.583} C_VEL
LIN {X 0,Y 390.765,Z 273.261,A -85,B 0,C 180,E1 17483.366,E2 17483.366} C_VEL
LIN {X 0,Y 387.601,Z 268.121,A -85,B 0,C 180,E1 17481.966,E2 17481.966} C_VEL
LIN {X 0,Y 385.095,Z 264.214,A -85,B 0,C 180,E1 17480.817,E2 17480.817} C_VEL
LIN {X 0,Y 384.217,Z 262.841,A -85,B 0,C 180,E1 17480.409,E2 17480.409} C_VEL
LIN {X 0,Y 381.782,Z 259.327,A -85,B 0,C 180,E1 17479.268,E2 17479.268} C_VEL
LIN {X 0,Y 381.06,Z 257.627,A -85,B 0,C 180,E1 17478.829,E2 17478.829} C_VEL
LIN {X 0,Y 378.525,Z 254.756,A -85,B 0,C 180,E1 17477.684,E2 17477.684} C_VEL
LIN {X 0,Y 377.678,Z 252.286,A -85,B 0,C 180,E1 17476.931,E2 17476.931} C_VEL
LIN {X 0,Y 377.656,Z 251.985,A -85,B 0,C 180,E1 17473.629,E2 17473.629} C_VEL
LIN {X 0,Y 377.661,Z 251.98,A -85,B 0,C 180,E1 17469.602,E2 17469.602} C_VEL
LIN {X 0,Y 377.671,Z 251.975,A -85,B 0,C 180,E1 17465.622,E2 17465.622} C_VEL
LIN {X 0,Y 377.675,Z 251.974,A -85,B 0,C 180,E1 17461.518,E2 17461.518} C_VEL
LIN {X 0,Y 377.68,Z 251.986,A -85,B 0,C 180,E1 17457.573,E2 17457.573} C_VEL
LIN {X 0,Y 377.694,Z 251.999,A -85,B 0,C 180,E1 17453.464,E2 17453.464} C_VEL
LIN {X 0,Y 377.682,Z 251.992,A -85,B 0,C 180,E1 17449.321,E2 17449.321} C_VEL
LIN {X 0,Y 377.691,Z 251.973,A -85,B 0,C 180,E1 17445.278,E2 17445.278} C_VEL
LIN {X 0,Y 377.685,Z 251.97,A -85,B 0,C 180,E1 17441.158,E2 17441.158} C_VEL
LIN {X 0,Y 377.689,Z 251.988,A -85,B 0,C 180,E1 17437.099,E2 17437.099} C_VEL
LIN {X 0,Y 377.688,Z 252.002,A -85,B 0,C 180,E1 17432.914,E2 17432.914} C_VEL
LIN {X 0,Y 377.685,Z 251.988,A -85,B 0,C 180,E1 17428.771,E2 17428.771} C_VEL
LIN {X 0,Y 377.679,Z 251.976,A -85,B 0,C 180,E1 17424.628,E2 17424.628} C_VEL
LIN {X 0,Y 377.684,Z 251.972,A -85,B 0,C 180,E1 17420.554,E2 17420.554} C_VEL
LIN {X 0,Y 377.68,Z 251.978,A -85,B 0,C 180,E1 17416.502,E2 17416.502} C_VEL
LIN {X 0,Y 377.681,Z 251.983,A -85,B 0,C 180,E1 17412.388,E2 17412.388} C_VEL
LIN {X 0,Y 377.679,Z 251.985,A -85,B 0,C 180,E1 17408.28,E2 17408.28} C_VEL
LIN {X 0,Y 377.715,Z 252.222,A -85,B 0,C 180,E1 17405.525,E2 17405.525} C_VEL
LIN {X 0,Y 379.294,Z 255.907,A -85,B 0,C 180,E1 17404.403,E2 17404.403} C_VEL
LIN {X 0,Y 381.079,Z 257.818,A -85,B 0,C 180,E1 17403.617,E2 17403.617} C_VEL
LIN {X 0,Y 383.028,Z 261.692,A -85,B 0,C 180,E1 17402.526,E2 17402.526} C_VEL
LIN {X 0,Y 384.298,Z 263.172,A -85,B 0,C 180,E1 17401.988,E2 17401.988} C_VEL
LIN {X 0,Y 386.581,Z 267.342,A -85,B 0,C 180,E1 17400.832,E2 17400.832} C_VEL
LIN {X 0,Y 387.958,Z 269.743,A -85,B 0,C 180,E1 17400.171,E2 17400.171} C_VEL
LIN {X 0,Y 390.874,Z 274.72,A -85,B 0,C 180,E1 17398.84,E2 17398.84} C_VEL
LIN {X 0,Y 395.704,Z 283.128,A -85,B 0,C 180,E1 17396.73,E2 17396.73} C_VEL
LIN {X 0,Y 402.734,Z 296.285,A -85,B 0,C 180,E1 17393.794,E2 17393.794} C_VEL
LIN {X 0,Y 410.536,Z 312.269,A -85,B 0,C 180,E1 17390.681,E2 17390.681} C_VEL
LIN {X 0,Y 418.099,Z 329.493,A -85,B 0,C 180,E1 17387.745,E2 17387.745} C_VEL
LIN {X 0,Y 410.826,Z 385.021,A -85,B 0,C 180,E1 17383.441,E2 17383.441} C_VEL
LIN {X 0,Y 409.249,Z 399.242,A -85,B 0,C 180,E1 17382.384,E2 17382.384} C_VEL
LIN {X 0,Y 413.912,Z 449.436,A -85,B 0,C 180,E1 17380.51,E2 17380.51} C_VEL
LIN {X 0,Y 408.136,Z 587.497,A -85,B 0,C 180,E1 17377.812,E2 17377.812} C_VEL
LIN {X 0,Y 407.04,Z 595.172,A -85,B 0,C 180,E1 17377.747,E2 17377.747} C_VEL
LIN {X 0,Y 401.329,Z 615.613,A -85,B 0,C 180,E1 17377.9,E2 17377.9} C_VEL
LIN {X 0,Y 400.464,Z 622.2,A -85,B 0,C 180,E1 17377.833,E2 17377.833} C_VEL
LIN {X 0,Y 399.132,Z 643.716,A -85,B 0,C 180,E1 17377.29,E2 17377.29} C_VEL
LIN {X 0,Y 397.267,Z 664.029,A -85,B 0,C 180,E1 17376.509,E2 17376.509} C_VEL
LIN {X 0,Y 395.036,Z 682.83,A -85,B 0,C 180,E1 17375.521,E2 17375.521} C_VEL
LIN {X 0,Y 392.343,Z 701.722,A -85,B 0,C 180,E1 17374.24,E2 17374.24} C_VEL
LIN {X 0,Y 389.377,Z 719.556,A -85,B 0,C 180,E1 17372.721,E2 17372.721} C_VEL
LIN {X 0,Y 386.301,Z 736.25,A -85,B 0,C 180,E1 17370.966,E2 17370.966} C_VEL
LIN {X 0,Y 383.18,Z 751.922,A -85,B 0,C 180,E1 17368.955,E2 17368.955} C_VEL
LIN {X 0,Y 380.129,Z 766.444,A -85,B 0,C 180,E1 17366.684,E2 17366.684} C_VEL
LIN {X 0,Y 377.35,Z 779.356,A -85,B 0,C 180,E1 17364.223,E2 17364.223} C_VEL
LIN {X 0,Y 374.971,Z 790.616,A -85,B 0,C 180,E1 17361.592,E2 17361.592} C_VEL
LIN {X 0,Y 373.014,Z 800.179,A -85,B 0,C 180,E1 17358.824,E2 17358.824} C_VEL
LIN {X 0,Y 371.57,Z 807.929,A -85,B 0,C 180,E1 17355.986,E2 17355.986} C_VEL
LIN {X 0,Y 370.561,Z 814.024,A -85,B 0,C 180,E1 17353.06,E2 17353.06} C_VEL
LIN {X 0,Y 369.926,Z 818.432,A -85,B 0,C 180,E1 17350.091,E2 17350.091} C_VEL
LIN {X 0,Y 369.618,Z 821.193,A -85,B 0,C 180,E1 17347.076,E2 17347.076} C_VEL
LIN {X 0,Y 369.547,Z 822.315,A -85,B 0,C 180,E1 17343.929,E2 17343.929} C_VEL
LIN {X 0,Y 369.705,Z 821.714,A -85,B 0,C 180,E1 17340.871,E2 17340.871} C_VEL
LIN {X 0,Y 370.11,Z 819.34,A -85,B 0,C 180,E1 17337.732,E2 17337.732} C_VEL
LIN {X 0,Y 370.857,Z 815.387,A -85,B 0,C 180,E1 17334.765,E2 17334.765} C_VEL
LIN {X 0,Y 372.068,Z 809.439,A -85,B 0,C 180,E1 17331.691,E2 17331.691} C_VEL
LIN {X 0,Y 373.78,Z 801.734,A -85,B 0,C 180,E1 17328.734,E2 17328.734} C_VEL
LIN {X 0,Y 376.043,Z 792.168,A -85,B 0,C 180,E1 17325.88,E2 17325.88} C_VEL
LIN {X 0,Y 378.713,Z 781.074,A -85,B 0,C 180,E1 17323.227,E2 17323.227} C_VEL
LIN {X 0,Y 381.73,Z 768.644,A -85,B 0,C 180,E1 17320.805,E2 17320.805} C_VEL
LIN {X 0,Y 385.035,Z 754.576,A -85,B 0,C 180,E1 17318.551,E2 17318.551} C_VEL
LIN {X 0,Y 388.392,Z 739.541,A -85,B 0,C 180,E1 17316.567,E2 17316.567} C_VEL
LIN {X 0,Y 391.662,Z 723.71,A -85,B 0,C 180,E1 17314.844,E2 17314.844} C_VEL
LIN {X 0,Y 395.063,Z 705.517,A -85,B 0,C 180,E1 17313.236,E2 17313.236} C_VEL
LIN {X 0,Y 398.099,Z 686.701,A -85,B 0,C 180,E1 17311.91,E2 17311.91} C_VEL
LIN {X 0,Y 400.759,Z 666.934,A -85,B 0,C 180,E1 17310.834,E2 17310.834} C_VEL
LIN {X 0,Y 402.897,Z 646.614,A -85,B 0,C 180,E1 17310.021,E2 17310.021} C_VEL
LIN {X 0,Y 404.469,Z 625.221,A -85,B 0,C 180,E1 17309.449,E2 17309.449} C_VEL
LIN {X 0,Y 413.826,Z 451.13,A -85,B 0,C 180,E1 17305.831,E2 17305.831} C_VEL
LIN {X 0,Y 409.497,Z 396.956,A -85,B 0,C 180,E1 17303.538,E2 17303.538} C_VEL
LIN {X 0,Y 409.072,Z 389.617,A -85,B 0,C 180,E1 17303.173,E2 17303.173} C_VEL
LIN {X 0,Y 417.039,Z 339.017,A -85,B 0,C 180,E1 17299.142,E2 17299.142} C_VEL
LIN {X 0,Y 411.143,Z 324.854,A -85,B 0,C 180,E1 17296.385,E2 17296.385} C_VEL
LIN {X 0,Y 405.653,Z 313.052,A -85,B 0,C 180,E1 17293.687,E2 17293.687} C_VEL
LIN {X 0,Y 401.232,Z 304.256,A -85,B 0,C 180,E1 17291.353,E2 17291.353} C_VEL
LIN {X 0,Y 397.182,Z 296.492,A -85,B 0,C 180,E1 17288.979,E2 17288.979} C_VEL
LIN {X 0,Y 394.514,Z 291.699,A -85,B 0,C 180,E1 17287.28,E2 17287.28} C_VEL
LIN {X 0,Y 392.124,Z 287.314,A -85,B 0,C 180,E1 17285.56,E2 17285.56} C_VEL
LIN {X 0,Y 389.93,Z 283.606,A -85,B 0,C 180,E1 17283.822,E2 17283.822} C_VEL
LIN {X 0,Y 389.286,Z 282.355,A -85,B 0,C 180,E1 17283.239,E2 17283.239} C_VEL
LIN {X 0,Y 386.808,Z 278.471,A -85,B 0,C 180,E1 17280.888,E2 17280.888} C_VEL
LIN {X 0,Y 386.283,Z 277.125,A -85,B 0,C 180,E1 17280.148,E2 17280.148} C_VEL
LIN {X 0,Y 383.437,Z 273.182,A -85,B 0,C 180,E1 17276.112,E2 17276.112} C_VEL
LIN {X 0,Y 382.824,Z 271.578,A -85,B 0,C 180,E1 17273.852,E2 17273.852} C_VEL
LIN {X 0,Y 382.656,Z 271.425,A -85,B 0,C 180,E1 17269.765,E2 17269.765} C_VEL
LIN {X 0,Y 383.336,Z 272.328,A -85,B 0,C 180,E1 17267.497,E2 17267.497} C_VEL
LIN {X 0,Y 386.174,Z 276.971,A -85,B 0,C 180,E1 17262.988,E2 17262.988} C_VEL
LIN {X 0,Y 386.985,Z 277.766,A -85,B 0,C 180,E1 17262.249,E2 17262.249} C_VEL
LIN {X 0,Y 389.202,Z 281.945,A -85,B 0,C 180,E1 17260.021,E2 17260.021} C_VEL
LIN {X 0,Y 390.47,Z 283.336,A -85,B 0,C 180,E1 17259.149,E2 17259.149} C_VEL
LIN {X 0,Y 392.554,Z 287.227,A -85,B 0,C 180,E1 17257.538,E2 17257.538} C_VEL
LIN {X 0,Y 393.716,Z 288.812,A -85,B 0,C 180,E1 17256.819,E2 17256.819} C_VEL
LIN {X 0,Y 396.979,Z 294.451,A -85,B 0,C 180,E1 17254.808,E2 17254.808} C_VEL
LIN {X 0,Y 401.818,Z 302.667,A -85,B 0,C 180,E1 17252.269,E2 17252.269} C_VEL
LIN {X 0,Y 407.414,Z 313.272,A -85,B 0,C 180,E1 17249.631,E2 17249.631} C_VEL
LIN {X 0,Y 413.263,Z 324.864,A -85,B 0,C 180,E1 17247.183,E2 17247.183} C_VEL
LIN {X 0,Y 417.956,Z 334.815,A -85,B 0,C 180,E1 17245.419,E2 17245.419} C_VEL
LIN {X 0,Y 422.267,Z 341.91,A -85,B 0,C 180,E1 17244.562,E2 17244.562} C_VEL
LIN {X 0,Y 422.903,Z 353.955,A -85,B 0,C 180,E1 17244.169,E2 17244.169} C_VEL
LIN {X 0,Y 416.519,Z 547.06,A -85,B 0,C 180,E1 17240.608,E2 17240.608} C_VEL
LIN {X 0,Y 413.191,Z 659.332,A -85,B 0,C 180,E1 17238.594,E2 17238.594} C_VEL
LIN {X 0,Y 411.385,Z 681.875,A -85,B 0,C 180,E1 17237.988,E2 17237.988} C_VEL
LIN {X 0,Y 408.99,Z 703.974,A -85,B 0,C 180,E1 17237.17,E2 17237.17} C_VEL
LIN {X 0,Y 406.152,Z 724.857,A -85,B 0,C 180,E1 17236.159,E2 17236.159} C_VEL
LIN {X 0,Y 402.666,Z 746.547,A -85,B 0,C 180,E1 17234.843,E2 17234.843} C_VEL
LIN {X 0,Y 398.94,Z 767.446,A -85,B 0,C 180,E1 17233.296,E2 17233.296} C_VEL
LIN {X 0,Y 395.004,Z 787.01,A -85,B 0,C 180,E1 17231.541,E2 17231.541} C_VEL
LIN {X 0,Y 390.68,Z 807.303,A -85,B 0,C 180,E1 17229.395,E2 17229.395} C_VEL
LIN {X 0,Y 386.702,Z 825.559,A -85,B 0,C 180,E1 17227.116,E2 17227.116} C_VEL
LIN {X 0,Y 382.943,Z 842.295,A -85,B 0,C 180,E1 17224.668,E2 17224.668} C_VEL
LIN {X 0,Y 379.429,Z 858.441,A -85,B 0,C 180,E1 17221.948,E2 17221.948} C_VEL
LIN {X 0,Y 376.36,Z 873.005,A -85,B 0,C 180,E1 17219.068,E2 17219.068} C_VEL
LIN {X 0,Y 373.542,Z 887.622,A -85,B 0,C 180,E1 17215.696,E2 17215.696} C_VEL
LIN {X 0,Y 371.522,Z 899.537,A -85,B 0,C 180,E1 17212.465,E2 17212.465} C_VEL
LIN {X 0,Y 370.08,Z 909.431,A -85,B 0,C 180,E1 17209.243,E2 17209.243} C_VEL
LIN {X 0,Y 369.14,Z 917.764,A -85,B 0,C 180,E1 17206.036,E2 17206.036} C_VEL
LIN {X 0,Y 368.587,Z 924.655,A -85,B 0,C 180,E1 17202.691,E2 17202.691} C_VEL
LIN {X 0,Y 368.313,Z 929.767,A -85,B 0,C 180,E1 17199.53,E2 17199.53} C_VEL
LIN {X 0,Y 368.257,Z 933.504,A -85,B 0,C 180,E1 17196.233,E2 17196.233} C_VEL
LIN {X 0,Y 368.241,Z 935.539,A -85,B 0,C 180,E1 17193.267,E2 17193.267} C_VEL
LIN {X 0,Y 368.246,Z 936.413,A -85,B 0,C 180,E1 17189.998,E2 17189.998} C_VEL
LIN {X 0,Y 368.235,Z 935.66,A -85,B 0,C 180,E1 17186.885,E2 17186.885} C_VEL
LIN {X 0,Y 368.235,Z 933.729,A -85,B 0,C 180,E1 17183.92,E2 17183.92} C_VEL
LIN {X 0,Y 368.295,Z 929.927,A -85,B 0,C 180,E1 17180.466,E2 17180.466} C_VEL
LIN {X 0,Y 368.565,Z 924.897,A -85,B 0,C 180,E1 17177.305,E2 17177.305} C_VEL
LIN {X 0,Y 369.119,Z 918.115,A -85,B 0,C 180,E1 17173.959,E2 17173.959} C_VEL
LIN {X 0,Y 370.066,Z 909.916,A -85,B 0,C 180,E1 17170.753,E2 17170.753} C_VEL
LIN {X 0,Y 371.611,Z 899.629,A -85,B 0,C 180,E1 17167.37,E2 17167.37} C_VEL
LIN {X 0,Y 373.568,Z 888.458,A -85,B 0,C 180,E1 17164.303,E2 17164.303} C_VEL
LIN {X 0,Y 376.287,Z 874.77,A -85,B 0,C 180,E1 17161.078,E2 17161.078} C_VEL
LIN {X 0,Y 379.387,Z 860.447,A -85,B 0,C 180,E1 17158.189,E2 17158.189} C_VEL
LIN {X 0,Y 382.999,Z 844.283,A -85,B 0,C 180,E1 17155.41,E2 17155.41} C_VEL
LIN {X 0,Y 386.925,Z 827.288,A -85,B 0,C 180,E1 17152.885,E2 17152.885} C_VEL
LIN {X 0,Y 390.909,Z 809.41,A -85,B 0,C 180,E1 17150.628,E2 17150.628} C_VEL
LIN {X 0,Y 395.288,Z 789.375,A -85,B 0,C 180,E1 17148.479,E2 17148.479} C_VEL
LIN {X 0,Y 399.354,Z 769.537,A -85,B 0,C 180,E1 17146.683,E2 17146.683} C_VEL
LIN {X 0,Y 402.976,Z 749.727,A -85,B 0,C 180,E1 17145.197,E2 17145.197} C_VEL
LIN {X 0,Y 406.464,Z 728.724,A -85,B 0,C 180,E1 17143.882,E2 17143.882} C_VEL
LIN {X 0,Y 409.501,Z 706.884,A -85,B 0,C 180,E1 17142.8,E2 17142.8} C_VEL
LIN {X 0,Y 412.125,Z 683.536,A -85,B 0,C 180,E1 17141.914,E2 17141.914} C_VEL
LIN {X 0,Y 414.018,Z 660.888,A -85,B 0,C 180,E1 17141.295,E2 17141.295} C_VEL
LIN {X 0,Y 416.137,Z 595.814,A -85,B 0,C 180,E1 17140.102,E2 17140.102} C_VEL
LIN {X 0,Y 422.525,Z 402.348,A -85,B 0,C 180,E1 17136.555,E2 17136.555} C_VEL
LIN {X 0,Y 424.198,Z 350.957,A -85,B 0,C 180,E1 17135.574,E2 17135.574} C_VEL
LIN {X 0,Y 423.415,Z 342.612,A -85,B 0,C 180,E1 17135.266,E2 17135.266} C_VEL
LIN {X 0,Y 414.234,Z 328.764,A -85,B 0,C 180,E1 17133.556,E2 17133.556} C_VEL
LIN {X 0,Y 405.391,Z 312.173,A -85,B 0,C 180,E1 17130.536,E2 17130.536} C_VEL
LIN {X 0,Y 397.711,Z 298.612,A -85,B 0,C 180,E1 17127.717,E2 17127.717} C_VEL
LIN {X 0,Y 392.132,Z 289.195,A -85,B 0,C 180,E1 17125.526,E2 17125.526} C_VEL
LIN {X 0,Y 388.454,Z 283.22,A -85,B 0,C 180,E1 17123.997,E2 17123.997} C_VEL
LIN {X 0,Y 386.19,Z 279.464,A -85,B 0,C 180,E1 17123.014,E2 17123.014} C_VEL
LIN {X 0,Y 383.077,Z 274.374,A -85,B 0,C 180,E1 17121.594,E2 17121.594} C_VEL
LIN {X 0,Y 380.034,Z 269.49,A -85,B 0,C 180,E1 17120.161,E2 17120.161} C_VEL
LIN {X 0,Y 377.376,Z 265.431,A -85,B 0,C 180,E1 17118.859,E2 17118.859} C_VEL
LIN {X 0,Y 376.551,Z 264.03,A -85,B 0,C 180,E1 17118.42,E2 17118.42} C_VEL
LIN {X 0,Y 374.15,Z 260.873,A -85,B 0,C 180,E1 17117.256,E2 17117.256} C_VEL
LIN {X 0,Y 372.924,Z 258.464,A -85,B 0,C 180,E1 17116.511,E2 17116.511} C_VEL
LIN {X 0,Y 370.559,Z 255.715,A -85,B 0,C 180,E1 17115.333,E2 17115.333} C_VEL
LIN {X 0,Y 369.749,Z 253.233,A -85,B 0,C 180,E1 17114.51,E2 17114.51} C_VEL
LIN {X 0,Y 369.706,Z 252.968,A -85,B 0,C 180,E1 17110.598,E2 17110.598} C_VEL
LIN {X 0,Y 369.704,Z 252.972,A -85,B 0,C 180,E1 17106.679,E2 17106.679} C_VEL
LIN {X 0,Y 369.708,Z 252.981,A -85,B 0,C 180,E1 17102.636,E2 17102.636} C_VEL
LIN {X 0,Y 369.712,Z 252.996,A -85,B 0,C 180,E1 17098.606,E2 17098.606} C_VEL
LIN {X 0,Y 369.716,Z 252.983,A -85,B 0,C 180,E1 17094.414,E2 17094.414} C_VEL
LIN {X 0,Y 369.717,Z 252.965,A -85,B 0,C 180,E1 17090.348,E2 17090.348} C_VEL
LIN {X 0,Y 369.72,Z 252.962,A -85,B 0,C 180,E1 17086.233,E2 17086.233} C_VEL
LIN {X 0,Y 369.724,Z 252.974,A -85,B 0,C 180,E1 17082.165,E2 17082.165} C_VEL
LIN {X 0,Y 369.73,Z 252.994,A -85,B 0,C 180,E1 17078.062,E2 17078.062} C_VEL
LIN {X 0,Y 369.735,Z 252.979,A -85,B 0,C 180,E1 17073.874,E2 17073.874} C_VEL
LIN {X 0,Y 369.733,Z 252.962,A -85,B 0,C 180,E1 17069.803,E2 17069.803} C_VEL
LIN {X 0,Y 369.733,Z 252.963,A -85,B 0,C 180,E1 17065.773,E2 17065.773} C_VEL
LIN {X 0,Y 369.738,Z 252.971,A -85,B 0,C 180,E1 17061.651,E2 17061.651} C_VEL
LIN {X 0,Y 369.74,Z 252.982,A -85,B 0,C 180,E1 17057.465,E2 17057.465} C_VEL
LIN {X 0,Y 369.743,Z 252.99,A -85,B 0,C 180,E1 17053.33,E2 17053.33} C_VEL
LIN {X 0,Y 369.751,Z 252.992,A -85,B 0,C 180,E1 17049.256,E2 17049.256} C_VEL
LIN {X 0,Y 369.795,Z 253.322,A -85,B 0,C 180,E1 17047.815,E2 17047.815} C_VEL
LIN {X 0,Y 371.294,Z 256.808,A -85,B 0,C 180,E1 17046.634,E2 17046.634} C_VEL
LIN {X 0,Y 373.325,Z 259.17,A -85,B 0,C 180,E1 17045.626,E2 17045.626} C_VEL
LIN {X 0,Y 375.115,Z 262.666,A -85,B 0,C 180,E1 17044.552,E2 17044.552} C_VEL
LIN {X 0,Y 376.679,Z 264.581,A -85,B 0,C 180,E1 17043.818,E2 17043.818} C_VEL
LIN {X 0,Y 378.82,Z 268.452,A -85,B 0,C 180,E1 17042.653,E2 17042.653} C_VEL
LIN {X 0,Y 379.986,Z 270.265,A -85,B 0,C 180,E1 17042.085,E2 17042.085} C_VEL
LIN {X 0,Y 383.122,Z 275.599,A -85,B 0,C 180,E1 17040.548,E2 17040.548} C_VEL
LIN {X 0,Y 388.387,Z 284.752,A -85,B 0,C 180,E1 17038.108,E2 17038.108} C_VEL
LIN {X 0,Y 395.554,Z 298.06,A -85,B 0,C 180,E1 17034.971,E2 17034.971} C_VEL
LIN {X 0,Y 402.188,Z 311.456,A -85,B 0,C 180,E1 17032.204,E2 17032.204} C_VEL
LIN {X 0,Y 409.167,Z 326.751,A -85,B 0,C 180,E1 17029.399,E2 17029.399} C_VEL
LIN {X 0,Y 411.928,Z 333.414,A -85,B 0,C 180,E1 17028.289,E2 17028.289} C_VEL
LIN {X 0,Y 404.363,Z 388.752,A -85,B 0,C 180,E1 17023.952,E2 17023.952} C_VEL
LIN {X 0,Y 403.307,Z 398.482,A -85,B 0,C 180,E1 17023.236,E2 17023.236} C_VEL
LIN {X 0,Y 407.988,Z 450.618,A -85,B 0,C 180,E1 17021.247,E2 17021.247} C_VEL
LIN {X 0,Y 400.464,Z 622.2,A -85,B 0,C 180,E1 17017.833,E2 17017.833} C_VEL
LIN {X 0,Y 399.329,Z 629.868,A -85,B 0,C 180,E1 17017.756,E2 17017.756} C_VEL
LIN {X 0,Y 393.32,Z 649.058,A -85,B 0,C 180,E1 17017.759,E2 17017.759} C_VEL
LIN {X 0,Y 391.777,Z 656.525,A -85,B 0,C 180,E1 17017.565,E2 17017.565} C_VEL
LIN {X 0,Y 389.539,Z 676.321,A -85,B 0,C 180,E1 17016.624,E2 17016.624} C_VEL
LIN {X 0,Y 387.006,Z 694.596,A -85,B 0,C 180,E1 17015.487,E2 17015.487} C_VEL
LIN {X 0,Y 383.977,Z 713.044,A -85,B 0,C 180,E1 17014.033,E2 17014.033} C_VEL
LIN {X 0,Y 380.891,Z 729.714,A -85,B 0,C 180,E1 17012.409,E2 17012.409} C_VEL
LIN {X 0,Y 377.578,Z 746.068,A -85,B 0,C 180,E1 17010.457,E2 17010.457} C_VEL
LIN {X 0,Y 374.402,Z 760.795,A -85,B 0,C 180,E1 17008.318,E2 17008.318} C_VEL
LIN {X 0,Y 371.424,Z 774.056,A -85,B 0,C 180,E1 17005.988,E2 17005.988} C_VEL
LIN {X 0,Y 368.754,Z 785.887,A -85,B 0,C 180,E1 17003.463,E2 17003.463} C_VEL
LIN {X 0,Y 366.455,Z 796.286,A -85,B 0,C 180,E1 17000.738,E2 17000.738} C_VEL
LIN {X 0,Y 364.575,Z 805.208,A -85,B 0,C 180,E1 16997.811,E2 16997.811} C_VEL
LIN {X 0,Y 363.25,Z 812.231,A -85,B 0,C 180,E1 16994.843,E2 16994.843} C_VEL
LIN {X 0,Y 362.369,Z 817.522,A -85,B 0,C 180,E1 16991.835,E2 16991.835} C_VEL
LIN {X 0,Y 361.857,Z 821.151,A -85,B 0,C 180,E1 16988.781,E2 16988.781} C_VEL
LIN {X 0,Y 361.653,Z 823.142,A -85,B 0,C 180,E1 16985.675,E2 16985.675} C_VEL
LIN {X 0,Y 361.679,Z 823.48,A -85,B 0,C 180,E1 16982.507,E2 16982.507} C_VEL
LIN {X 0,Y 361.945,Z 822.17,A -85,B 0,C 180,E1 16979.452,E2 16979.452} C_VEL
LIN {X 0,Y 362.508,Z 819.242,A -85,B 0,C 180,E1 16976.403,E2 16976.403} C_VEL
LIN {X 0,Y 363.447,Z 814.772,A -85,B 0,C 180,E1 16973.445,E2 16973.445} C_VEL
LIN {X 0,Y 364.817,Z 808.661,A -85,B 0,C 180,E1 16970.52,E2 16970.52} C_VEL
LIN {X 0,Y 366.737,Z 800.769,A -85,B 0,C 180,E1 16967.632,E2 16967.632} C_VEL
LIN {X 0,Y 369.272,Z 790.769,A -85,B 0,C 180,E1 16964.747,E2 16964.747} C_VEL
LIN {X 0,Y 372.161,Z 779.56,A -85,B 0,C 180,E1 16962.143,E2 16962.143} C_VEL
LIN {X 0,Y 375.471,Z 766.603,A -85,B 0,C 180,E1 16959.686,E2 16959.686} C_VEL
LIN {X 0,Y 379.009,Z 752.146,A -85,B 0,C 180,E1 16957.436,E2 16957.436} C_VEL
